	(*═════════════════════════════════════════════════════════*)
	(*  External Systems and I/O    *)
	(*═════════════════════════════════════════════════════════*)
	controlfb_control_b_start                                  , (* BOOL *)
	controlfb_control_b_stop                                   , (* BOOL *)
	controlfb_control_b_shutdown                               , (* BOOL *)
	controlfb_control_b_Reset                                  , (* BOOL *)
	controlfb_control_b_SystemShutdown                         , (* BOOL *)
	controlfb_control_b_EMstop                                 , (* BOOL *)
	controlfb_control_b_ClearHistory                           , (* BOOL *)
	controlfb_control_b_ActivateSettings                       , (* BOOL *)
	controlfb_control_b_startDeHum                             , (* BOOL *)
	controlfb_Operation_inputgrid_b_SyncClose                  , (* BOOL *)
	controlfb_Operation_Genset_b_manualStart                   , (* BOOL *)
	controlfb_Operation_PSB_b_SyncClose                        , (* BOOL *)
	controlfb_Operation_charger_b_StartCharging                , (* BOOL *)
	controlfb_Operation_charger_b_ResetCharger                 , (* BOOL *)
	controlfb_Operation_system_r_NominalVoltage                , (* REAL *)
	controlfb_Operation_system_r_NominalFrequency              , (* REAL *)
	controlfb_Operation_system_r_Pset                          , (* REAL *)
	controlfb_Operation_system_r_Qset                          , (* REAL *)
	controlfb_Operation_system_r_PFset                         , (* REAL *)
	controlfb_Operation_system_b_PFsetEnable                   , (* BOOL *)
	controlfb_Operation_system_b_SounderMute                   , (* BOOL *)
	controlfb_Operation_system_b_SounderTest                   , (* BOOL *)
	controlfb_Operation_system_b_GenGridModeTrans              , (* BOOL *)
	controlfb_Operation_system_b_GridTakeOverEnable            , (* BOOL *)
	controlfb_Operation_parallel_b_DetectSlaves                , (* BOOL *)
	controlfb_Operation_parallel_r_ActivePowerSlave1           , (* REAL *)
	controlfb_Operation_parallel_r_ReactivePowerSlave1         , (* REAL *)
	controlfb_Operation_parallel_r_ActivePowerSlave2           , (* REAL *)
	controlfb_Operation_parallel_r_ReactivePowerSlave2         , (* REAL *)
	controlfb_Operation_BMS_b_ManualStartHVDC                  , (* BOOL *)
	controlfb_SoftSettings_inputgrid_PeakshaveMode             , (* ePeakshaveMode *)
	controlfb_SoftSettings_inputgrid_setpointTimeslot1_r_SocTarget, (* REAL *)
	controlfb_SoftSettings_inputgrid_setpointTimeslot1_r_IdleChargePower, (* REAL *)
	controlfb_SoftSettings_inputgrid_setpointTimeslot1_r_FeedInCurrentLimitSoft, (* REAL *)
	controlfb_SoftSettings_inputgrid_setpointTimeslot1_r_SupplyCurrentLimitSoft, (* REAL *)
	controlfb_SoftSettings_inputgrid_setpointTimeslot2_r_SocTarget, (* REAL *)
	controlfb_SoftSettings_inputgrid_setpointTimeslot2_r_IdleChargePower, (* REAL *)
	controlfb_SoftSettings_inputgrid_setpointTimeslot2_r_FeedInCurrentLimitSoft, (* REAL *)
	controlfb_SoftSettings_inputgrid_setpointTimeslot2_r_SupplyCurrentLimitSoft, (* REAL *)
	controlfb_SoftSettings_inputgrid_b_BreakerControl          , (* BOOL *)
	controlfb_SoftSettings_inputgrid_b_ReverseCTDirection      , (* BOOL *)
	controlfb_SoftSettings_inputgrid_ui_CTrange                , (* UINT *)
	controlfb_SoftSettings_inputgrid_r_VTratio                 , (* REAL *)
	controlfb_SoftSettings_inputgrid_b_GridCodesActive         , (* BOOL *)
	controlfb_SoftSettings_inputgrid_b_WeakGridInput           , (* BOOL *)
	controlfb_SoftSettings_inputgrid_breaker_AutoConnect       , (* BOOL *)
	controlfb_SoftSettings_inputgrid_breaker_ShutdownDisconnect, (* BOOL *)
	controlfb_SoftSettings_inputgrid_breaker_EMstopDisconnect  , (* BOOL *)
	controlfb_SoftSettings_inputgrid_breaker_CurrentLimitDisconnect, (* BOOL *)
	controlfb_SoftSettings_inputgrid_breaker_CurrentLimitRetries, (* BYTE *)
	controlfb_SoftSettings_inputgenset_b_AutoStartStop         , (* BOOL *)
	controlfb_SoftSettings_inputgenset_b_HydridMode            , (* BOOL *)
	controlfb_SoftSettings_inputgenset_b_EnableSchedule        , (* BOOL *)
	controlfb_SoftSettings_inputgenset_setpointTimeslot1_r_SoCStart, (* REAL *)
	controlfb_SoftSettings_inputgenset_setpointTimeslot1_r_SoCStop, (* REAL *)
	controlfb_SoftSettings_inputgenset_setpointTimeslot1_r_BatteryloadStart, (* REAL *)
	controlfb_SoftSettings_inputgenset_setpointTimeslot1_r_BatteryloadStop, (* REAL *)
	controlfb_SoftSettings_inputgenset_setpointTimeslot1_b_StartAtBatteryError, (* BOOL *)
	controlfb_SoftSettings_inputgenset_setpointTimeslot2_r_SoCStart, (* REAL *)
	controlfb_SoftSettings_inputgenset_setpointTimeslot2_r_SoCStop, (* REAL *)
	controlfb_SoftSettings_inputgenset_setpointTimeslot2_r_BatteryloadStart, (* REAL *)
	controlfb_SoftSettings_inputgenset_setpointTimeslot2_r_BatteryloadStop, (* REAL *)
	controlfb_SoftSettings_inputgenset_setpointTimeslot2_b_StartAtBatteryError, (* BOOL *)
	controlfb_SoftSettings_inputgenset_b_PSBExtGensetMonitoring, (* BOOL *)
	controlfb_SoftSettings_inputgenset_b_FreqProtectionEnable  , (* BOOL *)
	controlfb_SoftSettings_inputgenset_Generator_e_GensetMode  , (* eGensetMode *)
	controlfb_SoftSettings_inputgenset_Generator_b_GensetLoadshareLine, (* BOOL *)
	controlfb_SoftSettings_inputgenset_Generator_r_RatedPower  , (* REAL *)
	controlfb_SoftSettings_inputgenset_Generator_r_powerloadMax, (* REAL *)
	controlfb_SoftSettings_inputgenset_Generator_r_PowerloadMin, (* REAL *)
	controlfb_SoftSettings_inputgenset_Generator_r_PowerloadEff, (* REAL *)
	controlfb_SoftSettings_inputgenset_Generator_r_ramprate    , (* REAL *)
	controlfb_SoftSettings_inputgenset_Generator_ui_CooldownTime, (* UINT *)
	controlfb_SoftSettings_inputgenset_Generator_ui_WarmupTime , (* UINT *)
	controlfb_SoftSettings_inputgenset_Loadbank_b_Enable       , (* BOOL *)
	controlfb_SoftSettings_inputgenset_Loadbank_r_PowerRating  , (* REAL *)
	controlfb_SoftSettings_inputgenset_Loadbank_r_PowerStepSize, (* REAL *)
	controlfb_SoftSettings_PSB_PeakshaveMode                   , (* ePeakshaveMode *)
	controlfb_SoftSettings_PSB_setpointTimeslot1_r_SocTarget   , (* REAL *)
	controlfb_SoftSettings_PSB_setpointTimeslot1_r_IdleChargePower, (* REAL *)
	controlfb_SoftSettings_PSB_setpointTimeslot1_r_FeedInCurrentLimitSoft, (* REAL *)
	controlfb_SoftSettings_PSB_setpointTimeslot1_r_SupplyCurrentLimitSoft, (* REAL *)
	controlfb_SoftSettings_PSB_setpointTimeslot2_r_SocTarget   , (* REAL *)
	controlfb_SoftSettings_PSB_setpointTimeslot2_r_IdleChargePower, (* REAL *)
	controlfb_SoftSettings_PSB_setpointTimeslot2_r_FeedInCurrentLimitSoft, (* REAL *)
	controlfb_SoftSettings_PSB_setpointTimeslot2_r_SupplyCurrentLimitSoft, (* REAL *)
	controlfb_SoftSettings_PSB_b_BreakerControl                , (* BOOL *)
	controlfb_SoftSettings_PSB_b_ReverseCTDirection            , (* BOOL *)
	controlfb_SoftSettings_PSB_ui_CTrange                      , (* UINT *)
	controlfb_SoftSettings_PSB_r_VTratio                       , (* REAL *)
	controlfb_SoftSettings_system_b_EnableSchedule             , (* BOOL *)
	controlfb_SoftSettings_system_b_EnableTransportMode        , (* BOOL *)
	controlfb_SoftSettings_system_b_EcoModeEnable              , (* BOOL *)
	controlfb_SoftSettings_system_e_UgridPowerMode             , (* eUgridPowerMode *)
	controlfb_SoftSettings_system_e_NetcontactorMode           , (* eNetcontMode *)
	controlfb_SoftSettings_system_e_UgridPowerLimitingMode     , (* ePLM *)
	controlfb_SoftSettings_system_b_AutomaticSwitching         , (* BOOL *)
	controlfb_SoftSettings_system_b_AMF                        , (* BOOL *)
	controlfb_SoftSettings_system_r_FrequencyDroop             , (* REAL *)
	controlfb_SoftSettings_system_r_VoltageDroop               , (* REAL *)
	controlfb_SoftSettings_system_r_SocMin                     , (* REAL *)
	controlfb_SoftSettings_system_r_SocMax                     , (* REAL *)
	controlfb_SoftSettings_system_r_PDischargeLimit            , (* REAL *)
	controlfb_SoftSettings_system_r_PChargeLimit               , (* REAL *)
	controlfb_SoftSettings_system_r_AMax                       , (* REAL *)
	controlfb_SoftSettings_system_s_SystemName                 , (* STRING(18) *)
	controlfb_SoftSettings_system_s_SMSnumber                  , (* STRING(18) *)
	controlfb_SoftSettings_system_ScheduleTimeSlot1_b_active   , (* BOOL *)
	controlfb_SoftSettings_system_ScheduleTimeSlot1_usi_DayOfWeek, (* USINT *)
	controlfb_SoftSettings_system_ScheduleTimeSlot1_usi_HourOfDay, (* USINT *)
	controlfb_SoftSettings_system_ScheduleTimeSlot1_usi_MinuteOfHour, (* USINT *)
	controlfb_SoftSettings_system_ScheduleTimeSlot2_b_active   , (* BOOL *)
	controlfb_SoftSettings_system_ScheduleTimeSlot2_usi_DayOfWeek, (* USINT *)
	controlfb_SoftSettings_system_ScheduleTimeSlot2_usi_HourOfDay, (* USINT *)
	controlfb_SoftSettings_system_ScheduleTimeSlot2_usi_MinuteOfHour, (* USINT *)
	controlfb_SoftSettings_system_by_LEDbrightness             , (* BYTE *)
	controlfb_SoftSettings_setup_e_AcInputType                 , (* eAcInputType *)
	controlfb_SoftSettings_setup_b_MasterSlaveMode             , (* BOOL *)
	controlfb_SoftSettings_setup_b_PeakshaveBoxEnable          , (* BOOL *)
	controlfb_SoftSettings_setup_e_Gridmode                    , (* eGridmode *)
	controlfb_SoftSettings_setup_e_DcCouplingType              , (* eDCinputType *)
	controlfb_SoftSettings_setup_b_ExtGenset                   , (* BOOL *)
	controlfb_HardSettings_setup_e_ControlSource               , (* eControlSources *)
	controlfb_HardSettings_charger_r_PowerMax                  , (* REAL *)
	controlfb_HardSettings_parallel_b_MasterSlaveEnabled       , (* BOOL *)
	controlfb_HardSettings_parallel_b_UnitIsMaster             , (* BOOL *)
	controlfb_HardSettings_parallel_b_ShutdownOnCommError      , (* BOOL *)
	controlfb_HardSettings_parallel_b_EffiencyMode             , (* BOOL *)
	controlfb_HardSettings_parallel_r_VoltageDroop             , (* REAL *)
	controlfb_HardSettings_parallel_r_FrequencyDroop           , (* REAL *)
	controlfb_HardSettings_system_r_PDischargeLimit            , (* REAL *)
	controlfb_HardSettings_system_r_PChargeLimit               , (* REAL *)
	controlfb_HardSettings_system_r_SMax                       , (* REAL *)
	controlfb_HardSettings_system_r_Amax                       , (* REAL *)
	controlfb_HardSettings_system_e_EarthingSystem             , (* eEarthingSystems *)
	controlfb_HardSettings_system_a_ui_InputCurrentLimit_1     , (* UINT *)
	controlfb_HardSettings_system_a_ui_InputCurrentLimit_2     , (* UINT *)
	controlfb_HardSettings_system_a_ui_OutputCurrentLimit_1    , (* UINT *)
	controlfb_HardSettings_system_a_ui_OutputCurrentLimit_2    , (* UINT *)
	controlfb_HardSettings_system_a_ui_OutputCurrentLimit_3    , (* UINT *)
	Generator_CommunicationOK                                  , (* BOOL *)
	Generator_FuelLow                                          , (* BOOL *)
	Generator_FuelCritical                                     , (* BOOL *)
	Generator_bGenBreakerClosed                                , (* BOOL *)
	Generator_bMainBreakerClosed                               , (* BOOL *)
	Generator_bGenRunning                                      , (* BOOL *)
	Generator_bGenVoltFreqOK                                   , (* BOOL *)
	Generator_bMainsFailure                                    , (* BOOL *)
	Generator_eActiveGenMode                                   , (* eGenOperationMode *)
	Generator_bIslandModeActive                                , (* BOOL *)
	Generator_bAMFActive                                       , (* BOOL *)
	Generator_bPeakshaveActive                                 , (* BOOL *)
	Generator_bFixedPowerActive                                , (* BOOL *)
	Generator_ar_LineVoltage_AVG                               , (* REAL *)
	Generator_ar_LineVoltage_L1                                , (* REAL *)
	Generator_ar_LineVoltage_L2                                , (* REAL *)
	Generator_ar_LineVoltage_L3                                , (* REAL *)
	Generator_ar_PhaseVoltage_AVG                              , (* REAL *)
	Generator_ar_PhaseVoltage_L1                               , (* REAL *)
	Generator_ar_PhaseVoltage_L2                               , (* REAL *)
	Generator_ar_PhaseVoltage_L3                               , (* REAL *)
	Generator_ar_Frequency_AVG                                 , (* REAL *)
	Generator_ar_Frequency_L1                                  , (* REAL *)
	Generator_ar_Frequency_L2                                  , (* REAL *)
	Generator_ar_Frequency_L3                                  , (* REAL *)
	Generator_ar_Current_AVG                                   , (* REAL *)
	Generator_ar_Current_L1                                    , (* REAL *)
	Generator_ar_Current_L2                                    , (* REAL *)
	Generator_ar_Current_L3                                    , (* REAL *)
	Generator_ar_PowerFactor_AVG                               , (* REAL *)
	Generator_ar_ActivePower_AVG                               , (* REAL *)
	Generator_ar_ActivePower_L1                                , (* REAL *)
	Generator_ar_ActivePower_L2                                , (* REAL *)
	Generator_ar_ActivePower_L3                                , (* REAL *)
	Generator_ar_ReactivePower_AVG                             , (* REAL *)
	Generator_ar_ApparentPower_AVG                             , (* REAL *)
	HartingIO_b_DigitalInput1Active                            , (* BOOL *)
	HartingIO_b_DigitalInput2Active                            , (* BOOL *)
	HartingIO_b_GenLowFuel                                     , (* BOOL *)
	HartingIO_b_ExtSystemShutdownRequest                       , (* BOOL *)
	HartingIO_b_ExtEMstopOK                                    , (* BOOL *)
	HartingIO_b_ExtEMstopActive                                , (* BOOL *)
	last
) DINT;
END_TYPE

// ---- POUs/MonitoringControl/IoT/DUTS/eIoTCommVersion.TcDUT
{attribute 'qualified_only'}
{attribute 'strict'}
TYPE eIoTCommVersion :
(
	V1 := 0,
	V2 := 1
);
END_TYPE

// ---- POUs/MonitoringControl/IoT/DUTS/eLogType.TcDUT
{attribute 'qualified_only'}
TYPE eLogType :
(
	none := 0,
	nuc := 1,
	cloud := 2
)UINT;
END_TYPE

// ---- POUs/MonitoringControl/IoT/DUTS/eUpdate.TcDUT
{attribute 'qualified_only'}
TYPE eUpdate :
(
	Fast			:= 0,
	Slow			:= 1,
	OnChange 		:= 2, //Updates only of variable has changed from previous value, but additionaly exactly once at system startup.
	Daily			:= 3
)UINT;
END_TYPE

// ---- POUs/MonitoringControl/IoT/DUTS/e_ORAttributeType.TcDUT
{attribute 'qualified_only'}
{attribute 'strict'}
TYPE e_ORAttributeType :
(
	text := 0,
	number := 2,
	integer := 3,
	JSON := 4
);
END_TYPE

// ---- POUs/MonitoringControl/IoT/DUTS/ST_AutoProvisioning.TcDUT
TYPE ST_AutoProvisioning :
	STRUCT
		sType	: STRING;
		sRealm	: STRING;
		sError	: STRING;
	END_STRUCT
END_TYPE

// ---- POUs/MonitoringControl/IoT/DUTS/ST_IotProps.TcDUT
TYPE ST_IotProps :
STRUCT
	sName		: STRING;
	sValue		: STRING(2000);
	eUpdate 	: eUpdate;
	st_RW		: ST_RW;
	pAdress		: PVOID;
	diSize		: DINT;
	ClassType : __SYSTEM.TYPE_CLASS;
	bNumber		: BOOL;
	bJson		: BOOL;
END_STRUCT
END_TYPE

// ---- POUs/MonitoringControl/IoT/DUTS/ST_RW.TcDUT
TYPE ST_RW :
STRUCT
	ReadFromNUC : BOOL:= FALSE;//enabling Read and Write can create unintended behaviour, consider feedback var
	WriteToNUC: BOOL:=FALSE ; //enabling Read and Write can create unintended behaviour, consider feedback var
END_STRUCT
END_TYPE

// ---- POUs/MonitoringControl/IoT/DUTS/ST_Supervisor.TcDUT
TYPE ST_Supervisor :
	STRUCT
		DATA	: STRING;
		ERROR	: STRING;
	END_STRUCT
END_TYPE

// ---- POUs/MonitoringControl/IoT/DUTS/ST_VarBuffer.TcDUT
TYPE ST_VarBuffer :
STRUCT
	sValue 	  : STRING(2000);
	pAdress   : PVOID;
	diSize	  : DINT;  
	ClassType : __SYSTEM.TYPE_CLASS;
	bNumber   : BOOL;
END_STRUCT
END_TYPE

// ---- POUs/MonitoringControl/IoT/_Structs/ST_IoTDataHMI.TcDUT
TYPE ST_IoTDataHMI :
STRUCT
	Label 				: STRING;
	Varname				: eDataMappingVarNames;
	Unit				: STRING(20);
	LogType 			: eLogType; 
	LogInterval 		: eUpdate;
	b_IOTWriteAllowed	: BOOL;
END_STRUCT
END_TYPE

// ---- POUs/MonitoringControl/IoT/_Structs/ST_IotData_credits.TcDUT
TYPE ST_IotData_credits :
STRUCT
	TotalCredits 		: DINT := 100;
	RemainingCredits	: DINT;
	UsedCredits			: DINT;
END_STRUCT
END_TYPE

// ---- POUs/MonitoringControl/IoT/_Structs/st_IOT_params.TcDUT
TYPE st_IOT_params :
STRUCT
	b_controlEnable			: 	BOOL := FALSE;
	r_UpdateTimeFast		: 	REAL := 15; //seconds
	r_UpdateTimeSlow		: 	REAL := 60; //seconds
	IotCommVersion			: 	eIotCommVersion;
	DefaultLoggingBudget	:	UINT	:= 100;
END_STRUCT
END_TYPE

// ---- POUs/MonitoringControl/IoT/_Structs/ST_IOT_SentStateLog.TcDUT
TYPE ST_IOT_SentStateLog :
STRUCT
	bUpdate			: BOOL;
	bMessageSent	: BOOL;
	LastIndexSent	: INT;
	LastIndex		: INT;
END_STRUCT
END_TYPE

// ---- POUs/MonitoringControl/_Enums/eAcInputType.TcDUT
{attribute 'qualified_only'}
{attribute 'strict'}
TYPE eAcInputType :
(
	None 	:= 0,
	Grid 	:= 1,
	Genset	:= 2
);
END_TYPE

// ---- POUs/MonitoringControl/_Enums/eCapTestSTate.TcDUT
{attribute 'qualified_only'}
{attribute 'strict'}
TYPE eCapTestSTate :
(
	init 				:= 	0,
	WriteSerial			:=	1,
	WriteNameplateCap	:=	2,
	WriteDatetime		:=	3,
	StartSystem 		:= 	4,
	InitialCharge 		:= 	5,
	RestPeriod1			:= 	6,
	DischargeCycle 		:= 	7,
	RestPeriod2 		:= 	8,
	ChargeCycle 		:= 	9,
	RestPeriod3 		:= 	10,
	StopSystem  		:= 	11,
	done				:=	12
);
END_TYPE

// ---- POUs/MonitoringControl/_Enums/eControlSources.TcDUT
{attribute 'qualified_only'}
{attribute 'strict'}
{attribute 'to_string'}
TYPE eControlSources :
(
	Local 				:= 0,
	ExternalController 	:= 1,
	PowerNet			:= 2	
);
END_TYPE

// ---- POUs/MonitoringControl/_Enums/eDcInputType.TcDUT
{attribute 'qualified_only'}
{attribute 'strict'}
TYPE eDcInputType :
(
	None := 0,
	Dc_charger := 1, 
	Dc_extender := 2
);
END_TYPE

// ---- POUs/MonitoringControl/_Enums/eEarthingSystems.TcDUT
{attribute 'qualified_only'}
{attribute 'strict'}
TYPE eEarthingSystems :
(
	None 		:= 0,	
	TN			:= 1,
	TN_ext		:= 2,
	IT			:= 3		
);
END_TYPE

// ---- POUs/MonitoringControl/_Enums/eGridFormingMode.TcDUT
{attribute 'qualified_only'}
{attribute 'strict'}
TYPE eGridFormingMode:
(
	Island := 0,
	Droop := 1
);
END_TYPE

// ---- POUs/MonitoringControl/_Enums/eGridMode.TcDUT
{attribute 'qualified_only'}
{attribute 'strict'}
{attribute 'to_string'}
TYPE eGridMode :
(
	auto := 0,
	following := 1,
	forming	:= 2
);
END_TYPE

// ---- POUs/MonitoringControl/_Enums/eNetContactorDirection.TcDUT
{attribute 'qualified_only'}
{attribute 'strict'}
TYPE eNetContactorDirection :
(
	Left 	:= -1,
	None 	:= 0,
	Right 	:= 1
);
END_TYPE

// ---- POUs/MonitoringControl/_Enums/eOperationMode.TcDUT
{attribute 'qualified_only'}
{attribute 'strict'}
TYPE eOperationMode :
(
	Auto := 0,
	Gridfollowing := 1,
	GridForming	:= 2
);
END_TYPE

// ---- POUs/MonitoringControl/_Enums/ePeakshaveMode.TcDUT
{attribute 'qualified_only'}
{attribute 'strict'}
TYPE ePeakshaveMode :
(
	Multiphase := 0,
	Singlephase := 1
);
END_TYPE

// ---- POUs/MonitoringControl/_Enums/ePowerControlType.TcDUT
{attribute 'qualified_only'}
{attribute 'strict'}
{attribue 'to_string}
TYPE ePowerControlType :
(
	Current := 0,
	Power	:=1,
	Both	:= 2
);
END_TYPE

// ---- POUs/MonitoringControl/_Enums/eSchedulerMode.TcDUT
{attribute 'qualified_only'}
{attribute 'strict'}
TYPE eSchedulerMode :
(
	continous := 0,
	daily := 1,
	weekly := 2
);
END_TYPE

// ---- POUs/MonitoringControl/_Enums/eSystemState.TcDUT
{attribute 'qualified_only'}
{attribute 'strict'}
{attribute 'to_string'}
TYPE eSystemState :
(
	Off 			:= 0,
	Shutdown 		:= 1,
	StandBy 		:= 2,
	Conditioning 	:= 3,
	Starting		:= 4,
	Running			:= 5,
	Charging_Only	:= 6,
	Discharging_Only:= 7,
	Stopped			:= 8,
	EMstop			:= 9,
	Reset			:= 10,
	Init			:= 11,
	Transport		:= 12,
	Dehumidifying	:= 13
);
END_TYPE

// ---- POUs/MonitoringControl/_Enums/eUgridPowerMode.TcDUT
{attribute 'qualified_only'}
{attribute 'strict'}
{attribute 'to_string'}
TYPE eUgridPowerMode :
(
	auto 			:= 0,
	DroopZeroStart	:= 1,
	Droop			:= 2,
	Isochronous		:= 3,
	None			:= 4
);
END_TYPE

// ---- POUs/MonitoringControl/_Structs/ST_ExtController_Events.TcDUT
TYPE ST_ExtController_Events :
STRUCT
	b_HeartbeatFault			: BIT;
	b_couplerError				:	bit;
	
	// control limit warnings
	b_FeedInLimitOutOfRange		: BIT;
	b_SupplyLimitOutOfRange 	: BIT;
	b_IdleChargePowerOutofRange	: BIT;
	b_BatOloadStartOutOfRange	: BIT;
	b_BatOloadStopOutOfRange	: BIT;
	b_SocTargetOutOfRange		: BIT;
	b_SocStartOutOfRange		: BIT;
	b_SocStopOutOfRange			: BIT;
	b_PsetOutOfRange			: BIT;
	b_QsetOutOfRange			: BIT;
	b_PFsetOutOfRange			: BIT;
	b_NominalVoltageOutOfRange	: BIT;
	b_NominalFreqOutOfRange		: BIT;
	b_FreqDroopOutOfRange		: BIT;
	b_VoltageDroopOutOfRange	: BIT;
	b_PmaxOutOfRange			: BIT;
	b_PminOutOfRange			: BIT;
	b_SmaxOutOfRange			: BIT;
	b_AmaxOutOfRange			: BIT;
	b_PowerRamprateOutOfRange	: BIT;
	b_PSBFeedInLimitOutOfRange	: BIT;
	b_PSBSupplyLimitOutOfRange: BIT;
	b_PSBIdleChargePowerOutOfRange: BIT;
	b_PSBSoCTargetOutOfRange	: BIT;
	b_SoCHighLimitOutOfRange	: BIT;
	b_SoCLowLimitOutOfRange		: BIT;
	b_GridModeValueOutOfRange	: BIT;
	b_PowermodeValueOutOfRange	: BIT;

END_STRUCT
END_TYPE

// ---- POUs/MonitoringControl/_Structs/ST_ExtController_get.TcDUT
TYPE ST_ExtController_get :
STRUCT
	control							: ST_ControlVars;
	Operation						: ST_OperationVars;
	SoftSettings					: ST_SoftSettings;
	HardSettings					: ST_HardSettings;
	events							: ST_ExtController_Events;
	b_AdvancedControl				: BOOL;
	ui_Heartbeat					: UINT;
	s_dashboardID					: STRING;
	b_Active						: BOOL;
	e_ConnectionState				: eConnectionState;
	s_OutputJson					: STRING(2000);
	LoggingBudgetOK					: BOOL := TRUE;
END_STRUCT
END_TYPE

// ---- POUs/MonitoringControl/_Structs/ST_ExtController_limits.TcDUT
TYPE ST_ExtController_limits :
STRUCT
	r_InputCtLimit			: REAL := 800;
	r_InverterPowerLimit	: REAL := 360;
	r_InverterCurrentLimit	: REAL := 520;
	r_NominalVoltageMin		: REAL := 360;
	r_NominalVoltageMax		: REAL := 440;
	r_NominalFreqMin		: REAL := 47.5;
	r_NominalFreqMax		: REAL := 52.5;
	r_DroopMax				: REAL := 10; 
	r_PowerRampLimit		: REAL := 300; //%/s
	r_PSBCtLimit			: REAL := 4000;
END_STRUCT
END_TYPE

// ---- POUs/MonitoringControl/_Structs/ST_ExtController_Set.TcDUT
TYPE ST_ExtController_Set :
STRUCT
	b_available				: BOOL;
END_STRUCT
END_TYPE

// ---- POUs/MonitoringControl/_Structs/ST_PLCPersistentVars.TcDUT
TYPE ST_PLCPersistentVars :
STRUCT
	Hardsettings					: ST_HardSettings; 
	Softsettings					: ST_Softsettings;
END_STRUCT
END_TYPE

// ---- POUs/Objects/4Grouter/Struct/ST_router_service.TcDUT
TYPE ST_router_service :
STRUCT
END_STRUCT
END_TYPE

// ---- POUs/Objects/ACDCCharger/Structs/ST_ACDCCharger_Service.TcDUT
TYPE ST_ACDCCharger_Service :
STRUCT
END_STRUCT
END_TYPE

// ---- POUs/Objects/BMS/eNums/eBMS_Status.TcDUT
{attribute 'qualified_only'}
{attribute 'strict'}
{attribute 'to_string'} 
TYPE eBMS_Status :
(
	Init := 0,
	Normal := 1,
	FullCharge := 2,
	FullDischarge := 3,
	Warning := 4,
	Fault := 5,
	off := 6
);
END_TYPE

// ---- POUs/Objects/BMS/eNums/eHVDC_Powerstatus.TcDUT
{attribute 'qualified_only'}
{attribute 'strict'}
TYPE eHVDC_Powerstatus :
(
	OFF := 0,
	Precharging := 1,
	ON	:= 2	
);
END_TYPE

// ---- POUs/Objects/BMS/eNums/ePOUState.TcDUT
{attribute 'qualified_only'}
{attribute 'strict'}
TYPE ePOUState :
(
	OFF := 0,
	PowerUp := 1,
	Init := 2,
	Normal	:=	3,
	EMSTOP	:=	4,
	Shutdown := 5
);
END_TYPE

// ---- POUs/Objects/BMS/eNums/ePowerControl.TcDUT
{attribute 'qualified_only'}
{attribute 'strict'}
TYPE ePowerControl :
(
	Init := 0,
	Stay := 1,
	PowerOn := 2,
	PowerOff := 3
)word;
END_TYPE

// ---- POUs/Objects/BMS/eNums/ePowerOnStatus.TcDUT
{attribute 'qualified_only'}
{attribute 'strict'}
TYPE ePowerOnStatus :
(
	Off := 0,
	On	:= 1,
	PowerOn_Fault := 2,
	PowerOff_Fault := 3
)UINT;
END_TYPE

// ---- POUs/Objects/BMS/Structs/st_BMS_BatterySummary.TcDUT
TYPE st_BMS_BatterySummary EXTENDS st_MBMU_BatterySummary :
STRUCT
	r_ratedPower				: REAL;
	r_ratedCurrent				: REAL;
	r_ratedEnergyCapacity		: REAL;
	ui_CycleCount				: UINT;
	r_SOCScaled					: REAL;
	b_chargingAllowed			: BOOL;
	b_dischargingAllowed		: BOOL;
	r_RemainingDischargeEnergyNett: REAL;
	r_RemainingChargeEnergyNett	: REAL;
	r_maxVoltageEver	 		: REAL;
	r_maxChargeCurrentEver		: REAL;
	r_maxDischargeCurrentEver	: REAL;
END_STRUCT
END_TYPE

// ---- POUs/Objects/BMS/Structs/st_BMS_Events.TcDUT
TYPE st_BMS_Events :
STRUCT
	//sunspec error list
	b_COMMUNICATION_ERROR			:	BOOL;
	b_OVER_TEMP_ALARM				:	BOOL;
	b_OVER_TEMP_WARNING				:	BOOL;
	b_UNDER_TEMP_ALARM				:	BOOL;
	b_UNDER_TEMP_WARNING			:	BOOL;
	b_OVER_CHARGE_CURRENT_ALARM		:	BOOL;
	b_OVER_CHARGE_CURRENT_WARNING	:	BOOL;
	b_OVER_DISCHARGE_CURRENT_ALARM	:	BOOL;
	b_OVER_DISCHARGE_CURRENT_WARNING:	BOOL;
	b_OVER_VOLT_ALARM				:	BOOL;
	b_OVER_VOLT_WARNING				:	BOOL;
	b_UNDER_VOLT_ALARM				:	BOOL;
	b_UNDER_VOLT_WARNING			:	BOOL;
	b_UNDER_SOC_MIN_ALARM			:	BOOL;
	b_UNDER_SOC_MIN_WARNING			:	BOOL;
	b_OVER_SOC_MAX_ALARM			:	BOOL;
	b_OVER_SOC_MAX_WARNING			:	BOOL;
	b_VOLTAGE_IMBALANCE_WARNING		:	BOOL;
	b_TEMPERATURE_IMBALANCE_ALARM	:	BOOL;
	b_TEMPERATURE_IMBALANCE_WARNING	:	BOOL;
	b_CONTACTOR_ERROR				:	BOOL;
	b_FAN_ERROR						:	BOOL;
	b_GROUND_FAULT					:	BOOL;
	b_OPEN_DOOR_ERROR				:	BOOL;
	b_CURRENT_IMBALANCE_WARNING		:	BOOL;
	b_OTHER_ALARM					:	BOOL;
	b_OTHER_WARNING					:	BOOL;
	b_CONFIGURATION_ALARM			:	BOOL;
	b_CONFIGURATION_WARNING			:	BOOL;
	b_POWERONFAULT					: 	BOOL;
	b_POWEROFFFAULT					:	BOOL;
	b_DISCONNECTOR_OFF				: 	BOOL;
	
	b_SocLowLimitOutOfRange			:	BOOL;
	b_SocHighLimitOutOfRange		: 	BOOL;
	
	b_SBMUCommError					:	ARRAY [0..3] OF BOOL;	
	b_SBMUFailedToConnect			:	ARRAY [0..3] OF BOOL;

	(* old event list. Replaced by sunspec
	BMSWatchdogWarning				:	BOOL;
	BMSWatchdogError				:	BOOL;
	
	BMSWarningStatus				:	BOOL;
	BMSFaultStatus					:	BOOL;
	
	BMSPowerOnFault					:	BOOL;
	BMSPowerOffFault				:	BOOL;
	
	SOCLowWarning					: 	BOOL;
	OverVoltageWarning				:	BOOL;
	UnderVoltageWarning				:	BOOL;
	VoltageBalanceWarning			:	BOOL;
	
	OverTemperatureWarning			:	BOOL;
	UnderTemperatureWarning			:	BOOL;
	TemperatureDifferenceWarning	:	BOOL;
	
	OverCurrentWarning				:	BOOL;
	
	CommunicationWarning			:	BOOL;
	
	OverVoltageError				:	BOOL;
	UnderVoltageError				:	BOOL;
	OverTemperatureError			:	BOOL;
	UnderTemperatureError			:	BOOL;
	
	CSCError						:	BOOL;
	SBMUError						:	BOOL;
	MBMUError						:	BOOL;
	
	CommunicationError				:	BOOL;
	*)
END_STRUCT
END_TYPE

// ---- POUs/Objects/BMS/Structs/st_BMS_Get.TcDUT
TYPE st_BMS_Get :
STRUCT
	BatteryInfo					: st_BMS_BatterySummary;
	t_RemainingTimeToAutoCalibration : TIME;
	//detailed info	
	MBMU						:	st_MBMU_Status;
	SBMU						:	ARRAY[0..3] OF st_SBMU_Status;
	
	Events						:	st_BMS_Events;
END_STRUCT
END_TYPE

// ---- POUs/Objects/BMS/Structs/st_BMS_Params.TcDUT
TYPE st_BMS_Params :
STRUCT
	IP_BMS							:	STRING(16) := '192.168.1.60';
	r_SocHysteresis					:   REAL := 1; // % 
	r_InternalConditioningSoCMin	: 	REAL := 30;
	r_SoCAbsoluteMin				: 	REAL := 6; // unscaled value
	r_SoCAbsoluteMax				: 	REAL := 100; //unscaled value

	r_KwhperString					: REAL := 208; //
	r_CrateBattery					: REAL := 0.5; //C
	r_AhperString					: REAL := 306; //Ah	
	b_DisableSOCAlarm				: BOOL := FALSE;
	b_ResetPersistentVars			: BOOL := FALSE;
	b_forcePrecharging				: BOOL := FALSE;
	
	b_EnableAutoCalibration			: BOOL := TRUE;
	t_AutoCalibrationInterval 		: TIME := T#14D;
END_STRUCT
END_TYPE

// ---- POUs/Objects/BMS/Structs/ST_BMS_Service.TcDUT
TYPE ST_BMS_Service :
STRUCT
END_STRUCT
END_TYPE

// ---- POUs/Objects/BMS/Structs/st_BMS_Set.TcDUT
TYPE st_BMS_Set :
STRUCT
	b_enable	: BOOL := TRUE;
	r_SocMax	: REAL := 90;
	r_SocMin	: REAL := 10;
END_STRUCT
END_TYPE

// ---- POUs/Objects/BMS/Structs/st_MBMU_BatterySummary.TcDUT
TYPE st_MBMU_BatterySummary :
STRUCT
		//general
	b_BMSHeartBeatOK				:	BOOL;
	e_BMS_PowerOnStatus				:	ePowerOnStatus;
	e_BMS_Status					:	eBMS_Status;		

	r_SystemVoltage					:	REAL;
	r_SystemCurrent					:	REAL;
	r_SOC							:	REAL;
	r_SOH							:	REAL := 100;
	ar_CellVoltage					:	ARRAY[0..2] OF REAL;
	ar_CellTemperature				:	ARRAY[0..2] OF REAL;
	r_MaxChargeCurrentAllowed		:	REAL;
	r_MaxDischargeCurrentAllowed	:	REAL;
	r_MaxChargePowerAllowed			:	REAL;
	r_MaxDischargePowerAllowed		:	REAL;
	r_MaxSystemVoltageAllowed		:	REAL;
	r_MinSystemVoltageAllowed		:	REAL;
	
	r_SystemPower					:	REAL;
	r_ChargeSOE						:	REAL;
	r_DischargeSOE					:	REAL;
	
	r_RemainingChargeEnergy			:	REAL;
	r_RemainingDischargeEnergy		:	REAL;
	
	r_HistAccChargeEnergy			:	REAL;
	r_HistAccDischargeEnergy		:	REAL;
END_STRUCT	
END_TYPE

// ---- POUs/Objects/BMS/Structs/st_MBMU_Status.TcDUT
TYPE st_MBMU_Status :
STRUCT
	GeneralSBMUStatus			:	ARRAY [0..15] OF WORD;
	MBMUStatus					:	ARRAY [0..15] OF WORD;

	s_MBMU_SWVer				:	STRING(16);
	s_MBMU_HWVer				:	STRING(16);
	
	s_ETH_SWVer					:	STRING(32);
	r_ETH_HWVer					:	STRING(32);	
	
	by_NumberOfSubSystems		:	BYTE;
	DateTime					:	ARRAY[0..5] OF WORD;
	b_InsulationSwitchOpen		:	BOOL;
	
	BatteryStatus				:	st_MBMU_BatterySummary;
END_STRUCT
END_TYPE

// ---- POUs/Objects/BMS/Structs/st_SBMU_BatterySummary.TcDUT
TYPE st_SBMU_BatterySummary :
STRUCT
	r_SystemVoltage			:	REAL;
	r_SystemCurrent			:	REAL;
	r_SOC					:	REAL;
	r_SOH					:	REAL;
	ar_CellVoltage				:	ARRAY[0..2] OF REAL;
	ar_CellTemperature			:	ARRAY[0..2] OF REAL;
	r_MaxChargeCurrentAllowed		:	REAL;
	r_MaxDischargeCurrentAllowed	:	REAL;
	r_HistAccChargeEnergy			:	REAL;
	r_HistAccDischargeEnergy		:	REAL;
	
	//Gaan we hier uberhaupt iets mee doen?
	w_MaxVoltageCellLocation 	: 	WORD;//ARRAY[0..1] OF BYTE;
	w_MinVoltageCellLocation 	:	 WORD;//ARRAY[0..1] OF BYTE;
	w_MaxTempCellLocation 		: 	WORD;//ARRAY[0..1] OF BYTE;
	w_MinTempCellLocation 		: 	WORD;//ARRAY[0..1] OF BYTE;
END_STRUCT
END_TYPE

// ---- POUs/Objects/BMS/Structs/st_SBMU_Status.TcDUT
TYPE st_SBMU_Status :
STRUCT
	w_SystemWarning			:	WORD;
	SystemAlarm				:	ARRAY [0..2] OF WORD;
	
	b_PrechargeRelayClosed	:	BOOL;
	b_MainPosRelayClosed	:	BOOL;
	b_MainNegRelayClosed	:	BOOL;
	b_ControlBoxFanOn		:	BOOL;
	b_BalanceStatus			:	BOOL;
	b_DoorState				:	BOOL;	
	
	s_SBMU_SWVer			:	STRING(16);
	s_SBMU_HWVer			:	STRING(16);
	s_CSC_SWVer				:	STRING(16);
	s_CSC_HWVer				:	STRING(16);
	
	BatteryStatus			:	st_SBMU_BatterySummary;
END_STRUCT
END_TYPE

// ---- POUs/Objects/CoolingSystem/enums/eConditioningRequirement.TcDUT
{attribute 'qualified_only'}
{attribute 'strict'}
{attribute 'to_string'}
TYPE eConditioningRequirement :
(
	none := 0,
	Pumprequired		:=	1,
	HeatingRequired 	:= 	2,
	CoolingRequired 	:= 	3
);
END_TYPE

// ---- POUs/Objects/CoolingSystem/enums/eCoolingSystemState.TcDUT
{attribute 'qualified_only'}
{attribute 'strict'}
{attribute 'to_string'}
TYPE eCoolingSystemState :
(
	OFF 						:= 	0,
	Circulating					:=	1,
	ActiveCooling				:= 	2,
	ActiveHeating				:= 	3,
	EMSTOP						:=	5
)uint := OFF;
END_TYPE

// ---- POUs/Objects/CoolingSystem/enums/eHeatPumpMode.TcDUT
{attribute 'qualified_only'}
{attribute 'strict'}
{attribute 'to_string'}
TYPE eHeatPumpMode :
(
	Standby := 0,
	Cooling := 1,
	Heating := 2
)UINT := Standby;
END_TYPE

// ---- POUs/Objects/CoolingSystem/enums/eHeatPumpState.TcDUT
{attribute 'qualified_only'}
{attribute 'strict'}
{attribute 'to_string'}
TYPE eHeatPumpState :
(
	OFF := 0,
	Initializing := 1,
	Standby := 2,
	Active_Cooling := 3,
	Active_Heating := 4,
	ERROR := 5
)UINT := OFF;
END_TYPE

// ---- POUs/Objects/CoolingSystem/enums/eSupportedHeatpumps.TcDUT
{attribute 'qualified_only'}
{attribute 'strict'}
TYPE eSupportedHeatpumps :
(
	TranePicco := 0,
	LgThermaV	:= 1
);
END_TYPE

// ---- POUs/Objects/CoolingSystem/structs/LG_Coils.TcDUT
TYPE LG_Coils :
STRUCT
	b_EnableOperation			:	BOOL := FALSE;
	b_EnableSwwOperation		: 	BOOL := FALSE;
	b_EnableSilentMode			:	BOOL := FALSE;
	b_EnableDesinfectionMode	:	BOOL := FALSE;
	b_EmstopActive				:	BOOL := FALSE;
	b_EnableEmStop				:	BOOL := FALSE;
END_STRUCT
END_TYPE

// ---- POUs/Objects/CoolingSystem/structs/LG_ControlRegs.TcDUT
TYPE LG_ControlRegs :
STRUCT
	ui_OperatingMode	:	UINT := 3;
	ui_ControlMode		:	UINT := 1;
	r_Setpoint1			:	REAL := 20;
	r_RoomSetpoint		:	REAL;
	ui_TempShiftValue	:	UINT;
	r_setpoint2			:	REAL;
	r_RoomSetpoint2		:	REAL;
	ui_TempShiftValue2	:	UINT;
	r_DHWgoalTemp		:	REAL;
	ui_EnergyStatus		:	UINT := 2;	
END_STRUCT
END_TYPE

// ---- POUs/Objects/CoolingSystem/structs/LG_InputRegs.TcDUT
TYPE LG_InputRegs :
STRUCT
	UI_ErrorCode		:	UINT;
	ui_OperationalMode	:	UINT;
	r_CoolantInletTemp	:	REAL;
	r_CoolantOutletTemp	:	REAL;
	r_BackupHeaterTemp	:	REAL;
	r_SWWTankTemp		:	REAL;
	r_SolarCollectorTemp:	REAL;
	r_RoomTemp1			:	REAL;
	r_FlowRate			:	REAL;
	r_FlowTempCircuit2	:	REAL;
	r_RoomTemp2			:	REAL;
	UI_EnergyStatus		:	UINT;
	r_OutsideTemp		:	REAL;	
	r_CoolantPressure	: Real;
END_STRUCT
END_TYPE

// ---- POUs/Objects/CoolingSystem/structs/LG_Statusbits.TcDUT
TYPE LG_Statusbits :
STRUCT
	b_WaterFlowNOK				:	BOOL;
	b_WaterPumpOn				:	BOOL;
	b_ExtWaterPumpOn			:	BOOL;
	b_CompressorOn				:	BOOL;
	b_DefrostOn					:	BOOL;
	b_SWWModeOn					:	BOOL;
	b_SWWTankDesinfectionActive	:	BOOL;
	b_SilentModeOn				:	BOOL;
	b_CoolingActive				:	BOOL;
	b_SolarPumpActive			:	BOOL;
	b_BackupHeater1Active		:	BOOL;
	b_BackupHeater2Active		:	BOOL;
	b_SWWBoostHeaterActive		:	BOOL;
	b_ErrorActive				:	BOOL;
	b_EMOperationAvailable		:	BOOL;
	b_EMSWWOperationAvailable	:	BOOL;
	b_MixPumpActive				:	BOOL;
	
END_STRUCT
END_TYPE

// ---- POUs/Objects/CoolingSystem/structs/ST_CoolingSystem_Events.TcDUT
TYPE ST_CoolingSystem_Events :
STRUCT
	//faults
	b_CoolingSystemFuseFailure		: 	BOOL;
	
	
	//System pressure dropped below idle minimum pressure. suspect coolant loss.
	b_CoolingLoopPressureLow	: 	BOOL := FALSE;	
	b_CoolingLoopPressureTooLow	: 	BOOL := FALSE;	
	
	//Temperature errors
	b_CoolantTempLow				: 	BOOL;
	b_CoolantTempTooHigh			: 	BOOL;
	b_CoolantTempHigh				: 	BOOL;
	
	HeatpumpEvents					:	ST_HeatpumpEvents;
END_STRUCT
END_TYPE

// ---- POUs/Objects/CoolingSystem/structs/ST_CoolingSystem_Get.TcDUT
TYPE ST_CoolingSystem_Get :
STRUCT
	CoolingSystemState		:	eCoolingSystemState;
	HeatPumpStatus			: 	eHeatPumpState;
	r_CoolantTemperature	:	REAL;
	r_CoolantPressure		:	REAL;
	r_EnclosureDewpoint		:	REAL;
	ui_DehumRemainingTime	: 	UINT; //minutes
	
	Heatpump			:	st_Heatpump_get;
	
	Events					: ST_CoolingSystem_Events;
END_STRUCT
END_TYPE

// ---- POUs/Objects/CoolingSystem/structs/ST_CoolingSystem_MaintenanceParams.TcDUT
TYPE ST_CoolingSystem_MaintenanceParams :
STRUCT
	//manual activation of cooling system. Max runtime is limited to 30 minutes
	b_ActivateCooling							: BOOL; 
	b_ActivateHeating							: BOOL;	
	
	
END_STRUCT
END_TYPE

// ---- POUs/Objects/CoolingSystem/structs/ST_Coolingsystem_params.TcDUT
TYPE ST_Coolingsystem_params :
STRUCT
	b_DoubleHeatpump							: BOOL := FALSE;
	
	// Minimum base coolant pressure
	r_MinimumSystemBasePressureWarningLevel		: REAL := 1;
	r_MinimumSystemBasePressureErrorLevel		: REAL := 0.7;

	PrimaryHeatpumpAddr							:	BYTE := 1;
	CoilSettings								:	BYTE := 2#0000_0001;
	SecondaryHeatpumpAddr						:	BYTE := 2;
	dw_HeatpumpOperationDelay					: DWORD := 30; // minutes
	
	//If the heatpump has run within this timeframe, no preheating is required before operation can start
	i_SkipHPPreheatingTime						: 	INT		:= 60; //minutes. 
	r_MinimumCoolantTemperatureForHPHeatingMode	:	REAL	:= 15;
	
	IO_IPaddress								: 	STRING := '192.168.1.52';
END_STRUCT
END_TYPE

// ---- POUs/Objects/CoolingSystem/structs/ST_HeatpumpData.TcDUT
TYPE ST_HeatpumpData :
STRUCT
	i_FW_Version		:	INT;		//1
	i_FW_release		:	INT;		//2
	w_FW_Subrelease		:	WORD;		//3
	w_FW_creationDate	:	WORD;		//4
	
	w_Serialnumber		:	ARRAY[0..17] OF WORD;	//80-97
	
	i_OperatingHours	:	INT;		//305-317?
	
	r_CoolantPower		:  	REAL;
	r_InletWaterTemp	:	REAL;		//400
	r_OutletWaterTemp	:	REAL;		//401
	r_HighPressure		:	REAL;		//406
	r_LowPressure		:	REAL;		//414
	r_CompInputTemp		:	REAL;		//422
	r_OutdoorTemp		:	REAL;		//428
	r_CompOutputTemp	:	REAL;		//433-435
	ui_WaterFlowRate		:	UINT;		//444
	
	w_ErrorList			:	ARRAY[1..7] OF WORD;	//950-956	
	
	r_FanSpeedPCT		:	REAL;		//7000
	r_PumpSpeedPCT		:	REAL;		//7001
	
	r_SetpointHeating	:	REAL;		//7204
	r_SetpointCooling	:	REAL;		//7203
	b_DefrostingActive	:	BOOL;		//7214.14
	
	HeatpumpEvents		:	st_HeatpumpEvents;
END_STRUCT
END_TYPE

// ---- POUs/Objects/CoolingSystem/structs/ST_HeatPumpEvents.TcDUT
TYPE ST_HeatPumpEvents :
STRUCT
	b_CommWarning		: BOOL;
	b_ProbeError		: BOOL;
	b_PressureError		: BOOL;
	b_CompressorError	: BOOL;
	b_ValveError		: BOOL;
	b_FanError			: BOOL;
	b_PumpError			: BOOL;
	b_WaterTempError	: BOOL;
	b_IOError			: BOOL;
	b_DefrostingActive	:	Bool;
	b_HeatpumpPreheatingActive	:	BOOL;
	b_TooColdForHeatpumpHeating	:	Bool;
END_STRUCT
END_TYPE

// ---- POUs/Objects/CoolingSystem/structs/ST_HeatPump_Get.TcDUT
TYPE ST_HeatPump_Get :
STRUCT
	HeatPumpState 	: 	eHeatPumpState;
	Setpoint		:	REAL;
	Events			: 	ST_HeatPumpEvents;
	
	HeatpumpData	:	ST_HeatpumpData;
END_STRUCT
END_TYPE

// ---- POUs/Objects/CoolingSystem/structs/st_TCME31_get_1.TcDUT
TYPE st_TCME31_get_1 :
STRUCT
	DigitalInput1	:	Bool;
	DigitalInput2	:	Bool;
	
	AnalogInput1	:	real;
	AnalogInput2	:	real;

	DigitalOutput1	:	Bool;
	DigitalOutput2	:	Bool;
	DigitalOutput3	:	Bool;
	DigitalOutput4	:	Bool;
	
	b_CommFault		:	Bool;
END_STRUCT
END_TYPE

// ---- POUs/Objects/CoolingSystem/structs/st_TCME31_Set_1.TcDUT
TYPE st_TCME31_Set_1 :
STRUCT
	IPAddress		:	String := '192.168.1.70';
	
	DigitalOutput1	:	Bool;
	DigitalOutput2	:	Bool;
	DigitalOutput3	:	Bool;
	DigitalOutput4	:	Bool;
END_STRUCT
END_TYPE

// ---- POUs/Objects/DCLink/_Enums/eDcLinkState.TcDUT
{attribute 'qualified_only'}
{attribute 'strict'}
{attribute 'to_string'} 

TYPE eDcLinkState :
(
	Disabled 	:= 0,
	Enabled	 	:= 1,
	Fault	 	:= 2
);
END_TYPE

// ---- POUs/Objects/DCLink/_Enums/eDCpowerPriority.TcDUT
{attribute 'qualified_only'}
{attribute 'strict'}
TYPE eDCpowerPriority :
(
	auto := 0,
	Inverter := 1,
	DCcoupling	:= 2
);
END_TYPE

// ---- POUs/Objects/DCLink/_Structs/ST_Bourns_errors.TcDUT
TYPE ST_Bourns_errors :
STRUCT
	b_OvervoltageError		:	BOOL;
	b_OverCurrentError		:	BOOL;
	b_OverTemperatureError	:	BOOL; 
	b_EnergyOverflow		:	BOOL;
	b_DeviceFault			:	BOOL;
	b_CommFault				:	BOOL;
END_STRUCT
END_TYPE

// ---- POUs/Objects/DCLink/_Structs/ST_Bourns_Powerdata.TcDUT
TYPE ST_Bourns_Powerdata :
STRUCT
	Power			: REAL;
	Current			: REAL;
	Voltage			: REAL;
	Energy			: REAL;
	EnergyImport	: REAL;
	EnergyExport	: REAL;
	Temperature		: REAL;
	Charge			: BOOL;
END_STRUCT
END_TYPE

// ---- POUs/Objects/DCLink/_Structs/ST_DCLink_events.TcDUT
TYPE ST_DCLink_events :
STRUCT
	OvercurrentTrip			: BOOL;
	OvervoltageNOK			: BOOL;
END_STRUCT
END_TYPE

// ---- POUs/Objects/DCLink/_Structs/ST_DCLink_Get.TcDUT
TYPE ST_DCLink_Get :
STRUCT
	b_DCCouplingState				: BOOL;
	Powerdata						: REFERENCE TO ST_Bourns_Powerdata;
	r_ratedCurrent					: REAL;
	r_BattChargePowerLimit			: REAL;
	r_BattDischargePowerLimit		: REAL;
	
	r_ExportPowerLimit				: REAL;
	r_ExportCurrentLimit			: REAL;
	r_ImportPowerLimit				: REAL;
	r_ImportCurrentLimit			: REAL;
	events							: ST_DCLink_events;
END_STRUCT
END_TYPE

// ---- POUs/Objects/DCLink/_Structs/ST_DCLink_IO.TcDUT
TYPE ST_DCLink_IO :
STRUCT
	bMCCBOpen		AT %Q*: BOOL;
	bMCCBClose		AT %Q*: BOOL;
	bUVRfb			AT %I*: BOOL;
END_STRUCT
END_TYPE

// ---- POUs/Objects/DCLink/_Structs/ST_DCLink_params.TcDUT
TYPE ST_DCLink_params :
STRUCT
	RatedCurrent			: UINT 		:= 250;
	OvercurrentTripDelay	: TIME		:= T#2S;
	IP						: STRING 	:= '192.168.1.62';
	DCpowerControlHyst		: REAL 		:= 0.1;	
	AllowClosingOnDeadBus	:	BOOL	:= FALSE;
	DIWiredToPLC			:	BOOL	:=	TRUE;
END_STRUCT
END_TYPE

// ---- POUs/Objects/DCLink/_Structs/ST_DCLink_set.TcDUT
TYPE ST_DCLink_set :
STRUCT
	b_DCBusEnable			:	Bool;
//	b_MCCBclose				: BOOL;
//	b_MCCBopen				: BOOL;
	r_ChargePowerLimit		: REAL;
	r_DischargePowerLimit	: REAL;
	r_DCCRatedPower			: REAL; // of the external device
	r_PowerRampRate			: REAL;
	e_DCpowerPriority		: eDCpowerPriority := eDCpowerPriority.DCcoupling;
END_STRUCT
END_TYPE

// ---- POUs/Objects/DCLink/_Structs/st_Pixsys.TcDUT
TYPE st_Pixsys :
STRUCT
	b_DoEnable			: BOOL;	
	b_DoFeedbackOn 		: BOOL;
	b_Di1				: BOOL;
	b_Di2				: BOOL;		
END_STRUCT
END_TYPE

// ---- POUs/Objects/PowerQualityMonitor/_Enums/eACRotationState.TcDUT
{attribute 'qualified_only'}
{attribute 'strict'}
{attribute 'to_string'}
TYPE eACRotationState :
(
	Left := -1,
	None := 0,
	Right := 1
);
END_TYPE

// ---- POUs/Objects/PowerQualityMonitor/_Structs/ST_PowerMonitor_BESS.TcDUT
TYPE ST_PowerMonitor_BESS :
STRUCT
	e_ACrotationStatus			: 	eACrotationState;
	ar_Current					:	ARRAY [0..4] OF REAL;
	r_LineVoltage				: 	REAL;
	r_Frequency					: 	REAL;
	r_currentUnbalance			:	REAL;
	//Power
	r_ApparentPower				: 	REAL;
	r_ReactivePower				: 	REAL;
	r_ActivePower				: 	REAL;
	//Energy Consumed
	r_EnergyConsumed			:	REAL;
	
	//Energy Delivered
	r_EnergySupplied			:	REAL;
	
	r_PowerFactor 				:	REAL;
END_STRUCT
END_TYPE

// ---- POUs/Objects/PowerQualityMonitor/_Structs/ST_PowerMonitor_Events.TcDUT
TYPE ST_PowerMonitor_Events :
STRUCT
	b_MBCommWarning 		: BOOL;
	b_MBCommError 			: BOOL;
	b_MBTimeoutWarning 		: BOOL;
	b_EL3443Warning			: BOOL;
	b_EL3443Error		: BOOL;
	b_ACdirectionDataInvalid: BOOL;
END_STRUCT
END_TYPE

// ---- POUs/Objects/PowerQualityMonitor/_Structs/ST_PowerMonitor_get.TcDUT
TYPE ST_PowerMonitor_get :
STRUCT
	InputField			:	ST_PowerMonitor_InputField;	
	OutputField			:	ST_PowerMonitor_OutputField;
	CEE					:   ST_PQVoltageData;
	Inverter			: 	ST_PQVoltageData;
	events				:	ST_PowerMonitor_Events;
END_STRUCT
END_TYPE

// ---- POUs/Objects/PowerQualityMonitor/_Structs/ST_PowerMonitor_InputField.TcDUT
TYPE ST_PowerMonitor_InputField EXTENDS st_PQVoltageData:
STRUCT
	r_loadshare					: 	REAL;
	ACQuality					:	ST_PQGridQualityData;
	Powerlock					: 	ARRAY [1..2] OF st_PQVoltageData;
END_STRUCT
END_TYPE

// ---- POUs/Objects/PowerQualityMonitor/_Structs/ST_PowerMonitor_OutputField.TcDUT
TYPE ST_PowerMonitor_OutputField EXTENDS st_PQVoltageData:
STRUCT
	r_loadshare					: 	REAL;
	ACQuality					:	ST_PQGridQualityData;
	Powerlock					: 	ARRAY [1..3] OF ST_PQPowerData;
END_STRUCT
END_TYPE

// ---- POUs/Objects/PowerStack/NetContactor/_Structs/ST_Netcontactor_service.TcDUT
TYPE ST_Netcontactor_service :
STRUCT
	Right			: ST_service_DigitalOutInWithSafety;
	Left			: ST_service_DigitalOutInWithSafety;
END_STRUCT
END_TYPE

// ---- POUs/Objects/PowerStack/_Structs/ST_Powermodule_Service.TcDUT
TYPE ST_Powermodule_Service :
STRUCT
	b_FieldBusControlEnable			: BOOL := TRUE;
	b_FanOn							: eForceBool;
END_STRUCT
END_TYPE

// ---- POUs/Objects/PowerStack/_Structs/ST_Powerstack_MaintenanceParams.TcDUT
TYPE ST_Powerstack_MaintenanceParams :
STRUCT
	ForceNetcontactor		: BOOL;
END_STRUCT
END_TYPE

// ---- POUs/Objects/PowerStack/_Structs/ST_Powerstack_Service.TcDUT
TYPE ST_Powerstack_Service :
STRUCT
	Netcontactor			: St_Netcontactor_service;
	PowermoduleMaster		: ST_Powermodule_Service;
	PowermoduleSlave		: ST_Powermodule_Service;
END_STRUCT
END_TYPE

// ---- POUs/Safety/ST_Safety_ContactorEDM.TcDUT
TYPE ST_Safety_ContactorEDM :
STRUCT
	b_MccbMasterEDM						: BOOL;
	b_MccbSlaveEDM						: BOOL;
	b_NetcontactorEDM					: BOOL;
	b_DcMccbEDM							: BOOL;
END_STRUCT
END_TYPE

// ---- POUs/Safety/ST_Safety_get.TcDUT
TYPE ST_Safety_get :
STRUCT
	b_SafetyOK					: BOOL;
	b_SafetyDcOK				: BOOL;
	b_EstopChannelAOK			: BOOL;		
	b_EstopChannelBOK			: BOOL;		
	b_InsulationMonitorOK		: BOOL;	
	b_MRCDBOK					: BOOL;	
	b_InverterDoorOK            : BOOL;
	b_ZptOK				        : BOOL;
END_STRUCT
END_TYPE

// ---- POUs/Safety/ST_Safety_ToSafetyPrg.TcDUT
TYPE ST_Safety_ToSafetyPrg :
STRUCT
	b_ErrorReset						: BOOL;
	b_EmergencyStopSoftwareOK			: BOOL;
	b_SafetyRunStop						: BOOL := TRUE;
	contactors							: ST_Safety_ContactorEDM;
END_STRUCT
END_TYPE

// ---- POUs/Objects/4Grouter/Struct/dwtoreal.TcDUT
TYPE dwtoreal :
UNION
	Registers	:	ARRAY[1..2] OF WORD;
	dwordvalue	:	dword;
	realvalue	:	REAL;
END_UNION
END_TYPE

// ---- POUs/Objects/4Grouter/Struct/eModemState.TcDUT
{attribute 'qualified_only'}
//{attribute 'strict'}
TYPE eModemState :
(
	Disconnected := 0,
	Connected := 1
);
END_TYPE

// ---- POUs/Objects/4Grouter/Struct/eNetworkState.TcDUT
{attribute 'qualified_only'}
//{attribute 'strict'}
TYPE eNetworkState :
(
	unknown := 0,
	searching := 1,
	Unregistered := 2,
	Registered := 3,
	Roaming := 4
	);
END_TYPE

// ---- POUs/Objects/4Grouter/Struct/eSimSelectionMode.TcDUT
{attribute 'qualified_only'}
{attribute 'strict'}
TYPE eSimSelectionMode :
(
	auto := 0,
	force_sim1 := 1,
	force_sim2 := 2
);
END_TYPE

// ---- POUs/Objects/4Grouter/Struct/eSimState.TcDUT
{attribute 'qualified_only'}
//{attribute 'strict'}
TYPE eSimState :
(
	no_sim := 0,
	Inserted := 1,
	active := 2,
	pin_fault := 3
);
END_TYPE

// ---- POUs/Objects/4Grouter/Struct/eSMSStatus.TcDUT
{attribute 'qualified_only'}
//{attribute 'strict'}
TYPE eSMSStatus :
(
	Idle 			:= 	0,
	NewMessage 		:= 	1,
	SendingMessage 	:= 	2,
	error			:=	3
);
END_TYPE

// ---- POUs/Objects/4Grouter/Struct/eWifiSecurityTypes.TcDUT
{attribute 'qualified_only'}
{attribute 'strict'}
{attribute 'to_string'}
TYPE eWifiSecurityTypes :
(
	none := 0,
	PSK2 := 1,
	SAE  := 2,
	SAE_mixed := 3,
	PSK := 4	
);
END_TYPE

// ---- POUs/Objects/4Grouter/Struct/eWifiStatus.TcDUT
{attribute 'qualified_only'}
TYPE eWifiStatus :
(
	invalid := 0,
	off := 1,
	searching := 2,
	Connected := 3,
	Starting := 4,
	Active := 5
);
END_TYPE

// ---- POUs/Objects/4Grouter/Struct/st_Device.TcDUT
TYPE st_Device :
STRUCT
	SystemUptime	:	UDINT;	
	Temperature		:	REAL;
	RouterSerial	:	STRING(32);
END_STRUCT
END_TYPE

// ---- POUs/Objects/4Grouter/Struct/st_GPS.TcDUT
TYPE st_GPS :
STRUCT
	Latitude 	: 	REAL;
	Longitude 	: 	REAL;
	FixTime 	: 	STRING(32);
	DateTime	:	DT;
	Speed		:	REAL;
	SatCount	:	UINT;
	Accuracy	:	REAL;	
END_STRUCT
END_TYPE

// ---- POUs/Objects/4Grouter/Struct/st_mobile.TcDUT
TYPE st_mobile :
STRUCT
	NetworkOperator				:	STRING(32);
	NetworkInfo					:	STRING(32);
	NetworkType					:	STRING(32);
	RSSI						:	DINT;
	ui_Sim1DataSendMonth		:	UINT;
	ui_Sim1DataReceivedMonth	:	UINT;
	ui_Sim2DataSendMonth		:	UINT;
	ui_Sim2DataReceivedMonth	:	UINT;
	s_EmergencySMSNumber		:	STRING(20);
	s_SecondarySMSNumber		:	STRING(20);
	s_EmergencySMSDevName		:	STRING(18);
	st_LatestSMSMessage			:	STRING(80);
	ModemState					:	eModemState;
	NetworkState				:	eNetworkState;
	ui_ActiveSim				:	UINT;
	SimStatus					:	eSimState;
END_STRUCT
END_TYPE

// ---- POUs/Objects/4Grouter/Struct/st_Router_Events.TcDUT
TYPE st_Router_Events :
STRUCT
	b_MBCommWarning		:	BOOL;
	b_NoSimWarning		:	BOOL;
	b_NoNetworkWarning	: 	BOOL;
	b_noGPSFixWarning	:	BOOL;
	b_SMSNotSendError	:	BOOL; 
	b_NoSMSNumberAvailable	:	BOOL;
	b_TimeUpdateFailed 	: BOOL;
END_STRUCT
END_TYPE

// ---- POUs/Objects/4Grouter/Struct/st_router_get.TcDUT
TYPE st_router_get :
STRUCT
	Device 		: 	st_Device;
	GPS			:	st_GPS;
	Mobile		:	st_mobile;
	Wifi		:	st_Wifi;
	e_SMSStatus : 	eSMSStatus;
	Events		:	st_Router_Events;
END_STRUCT
END_TYPE

// ---- POUs/Objects/4Grouter/Struct/ST_Router_params.TcDUT
TYPE ST_Router_params :
STRUCT
	IP_TELTONIKA		: STRING(16) := '192.168.1.1';
	MBPort_TELTONIKA 	: UINT := 502;
	T_MBTimeout			: TIME := T#2S;
	MinimumPhoneNumberLength	:UINT := 10;
	
	//temporary setup via stparams until integrated into HMI
	ManualSettings		:	st_router_set;
END_STRUCT
END_TYPE

// ---- POUs/Objects/4Grouter/Struct/ST_Router_set.TcDUT
TYPE ST_Router_set :
STRUCT
	EnableWifiClient	:	BOOL;
	WifiClientSSID		:	STRING(32) := 'MachineAccessPoint@VDL';
	WifiClientPass		:	STRING(32) := 'e4ff1c12kLL';
	WifiClientSecType	:	eWifiSecurityTypes := eWifiSecurityTypes.PSK2;
	
	EnableWifiAP		:	BOOL;
	WifiAPSSID			:	STRING(32) := 'ePU10_AP';
	WifiAPPass			:	STRING(32) := 'Welkom!VDL';
	WifiAPSecType		:	eWifiSecurityTypes := eWifiSecurityTypes.PSK2;
	
	SimSelectionMode	:	eSimSelectionMode := eSimSelectionMode.auto;
	Sim1Pin				:	STRING(4) := '0000';
	Sim2Pin				:	STRING(4) := '0000';
	
	UpdateSystemTime	:	BOOL;
	
	AutoRebootEnable	:	BOOL;
	ManualReboot		:	BOOL;
END_STRUCT
END_TYPE

// ---- POUs/Objects/4Grouter/Struct/st_Wifi.TcDUT
TYPE st_Wifi :
STRUCT
	WifiClienModeStatus		:	eWifiStatus;
	WifiAPModeStatus		:	eWifiStatus;
	WifiApNumberOfClients	:	Uint;
END_STRUCT
END_TYPE

// ---- POUs/Objects/ACDCCharger/Enums/eAcDcChargerState.TcDUT
{attribute 'qualified_only'}
{attribute 'strict'}
{attribute 'to_string'} 

TYPE eAcDcChargerState :
(
	init 		:= 0,
	off 		:= 1,
	Standby	 	:= 2,
	starting 	:= 4,
	running		:=	5,
	stopping	:=	6, 

	fault 		:= 7
);
END_TYPE

// ---- POUs/Objects/ACDCCharger/Structs/Hadi/E_ChargerState.TcDUT
TYPE E_ChargerState :
(
    Idle := 0,
    ModulesOff := 10,
    SetVI := 20,
    CheckVoltage := 30,
    EnableModules := 40,
    Running := 100,
    Shutdown := 200,
    OpenRelay := 210,
    Fault := 900
);
END_TYPE

// ---- POUs/Objects/ACDCCharger/Structs/Hadi/ST_CanId.TcDUT
TYPE ST_CanId :
STRUCT
    ExtendedBit : BOOL;   // Bit31 (should always be TRUE)
    ErrorCode   : BYTE;   // Bits 28..26
    DeviceNo    : BYTE;   // Bits 25..22
    CommandNo   : BYTE;   // Bits 21..16
    TargetAddr  : BYTE;   // Bits 15..8
    SourceAddr  : BYTE;   // Bits 7..0
END_STRUCT
END_TYPE

// ---- POUs/Objects/ACDCCharger/Structs/Hadi/ST_ChargerControl.TcDUT
TYPE ST_ChargerControl :
STRUCT
    (* Charger control *)
    bStartCharge      : BOOL;   // start charging sequence
    bStopCharge       : BOOL;   // stop charging sequence

    (* Module enable command *)
    bEnableModules    : BOOL;   // CMD 1A

    (* Setpoints *)
    rSetVoltage       : REAL;   // desired voltage [V]
    rSetCurrent       : REAL;   // desired current [A]

    (* Apply commands *)
    bApplyGroupSet    : BOOL;   // CMD 1B (group control)
    bApplyModuleSet   : BOOL;   // CMD 1C (module control)

    (* Target module *)
    ModuleTarget      : BYTE;   // module number (peer-to-peer)

    (* Hardware relay *)
    bSystemRelayCmd   : BOOL;   // command to close system relay
END_STRUCT
END_TYPE

// ---- POUs/Objects/ACDCCharger/Structs/Hadi/ST_Control.TcDUT
TYPE ST_Control :
STRUCT
	rLimitInputCurrent	: REAL;	// CMD 0F Limit input current on all power modules
//	stModuleControl		: ARRAY [0..10] OF REAL;
	bEnableDisable		: BOOL; // CMD 1A (Broadcastong or Group)
	rSetOutputVoltage	: REAL;	// CMD 1B
	rSetOutputCurrent	: REAL;	// CMD 1B
	bResetMode			: BOOL;	// CMD 1E
	
END_STRUCT
END_TYPE

// ---- POUs/Objects/ACDCCharger/Structs/Hadi/ST_Data.TcDUT
TYPE ST_Data :
STRUCT
	rSystemOutVoltageDc		: REAL;		// CMD 01
	rSystemOutCurrentDc		: REAL;		// CMD 01
	rNumberOfModules		: REAL;		// CMD 02
	stModuleData			: ARRAY [0..10] OF ST_ModuleData;
	
	
	
	
	
END_STRUCT
END_TYPE

// ---- POUs/Objects/ACDCCharger/Structs/Hadi/ST_ModuleControl.TcDUT
TYPE ST_ModuleControl :
STRUCT
	bEnableDisable		: BOOL; // CMD 1A
	rSetOutputVoltage	: REAL;	// CMD 1C
	rSetOutputCurrent	: REAL;	// CMD 1C
	
	
	
	
END_STRUCT
END_TYPE

// ---- POUs/Objects/ACDCCharger/Structs/Hadi/ST_ModuleData.TcDUT
TYPE ST_ModuleData :
STRUCT
	rOutVoltageDc		: REAL;	// CMD 03
	rOutCurrentDc		: REAL;	// CMD 03
	rTemprature			: REAL;	// CMD 04
	rStatus0			: REAL;	// CMD 04
	rStatus1			: REAL;	// CMD 04
	rStatus2			: REAL;	// CMD 04
	rVoltageL1L2		: REAL;	// CMD 06
	rVoltageL2L3		: REAL;	// CMD 06
	rVoltageL3L1		: REAL;	// CMD 06
	rExternalVoltageDc	: REAL;	// CMD 0C      this could be the same as rOutVoltageDc CMD 03
	ravilableCurrentDc	: REAL;	// CMD 0C
	
	 stStatus           : ST_ModuleStatus;  // decoded status bits
	 
	 bValid		: BOOL; // validate if data are updating
	
END_STRUCT
END_TYPE

// ---- POUs/Objects/ACDCCharger/Structs/Hadi/ST_ModuleStatus.TcDUT
TYPE ST_ModuleStatus :
STRUCT
	 (* STATUS 2 *)
    bPfcOff              : BOOL;	// Bit 7
    bInputOverVoltage    : BOOL;	// Bit 6	
    bInputUnderVoltage   : BOOL;	// Bit 5
    bInputAsymmetry      : BOOL;	// Bit 4
    bPhaseLost           : BOOL;	// Bit 3
    bLoadSharingError    : BOOL;	// Bit 2
    bModuleIdDuplicate   : BOOL;	// Bit 1
    bPowerLimitation     : BOOL;	// Bit 0

    (* STATUS 1 *)
    bCanTimeout          : BOOL;	// Bit 7    /////////
    bSlowStartup         : BOOL;	// Bit 6
    bOutputOverVoltage   : BOOL;	// Bit 5
    bTempHigh            : BOOL;	// Bit 4
    bFanError            : BOOL;	// Bit 3
    bModuleProtection    : BOOL;	// Bit 2
    bModuleError         : BOOL;	// Bit 1      ////////////
    bDcSideOff           : BOOL;	// Bit 0

    (* STATUS 0 *)
    bDischargeAbnormal   : BOOL;	// Bit 5
    bMpptSwitchMode      : BOOL;	// Bit 4
    bPfcAbnormal         : BOOL;	// Bit 3
    bInternalCommError   : BOOL;	// Bit 2
    bOutputShortCircuit  : BOOL;	// Bit 0
END_STRUCT
END_TYPE

// ---- POUs/Objects/ACDCCharger/Structs/ST_ACDCCharger_events.TcDUT
TYPE ST_ACDCCharger_events :
STRUCT
	b_CommunicationFault			:	BOOL;
	b_BuscouplerNotFound			:	BOOL;
	b_ACUnderVoltageDeratingActive	: 	BOOL;
	b_BatteryLimitDeratingActive	:	BOOL;
	b_TemperatureDeratingActive		:	BOOL;
	b_CurrentLimitActive			:	BOOL;
	b_SOCLimitReached				:	BOOL;
	b_FailedToGenerateDCOutput		:	BOOL;
	B_ACPhaselossFault				:	BOOL;
	B_ACUndervoltage				:	BOOL;
	B_ACOvervoltage					:	BOOL;
END_STRUCT
END_TYPE

// ---- POUs/Objects/ACDCCharger/Structs/ST_ACDCCharger_get.TcDUT
TYPE ST_ACDCCharger_get :
STRUCT
	e_SystemStatus			: eAcDCChargerState := eACDCChargerState.init;
	
	by_NoModulesActive		: BYTE;	
	by_NoModulesInstalled	: BYTE;
	e_ChargerStatus 		: ARRAY [0..6] OF eAcDcChargerState;
	
	ar_ACvoltage			: ARRAY [0..3] OF REAL;
	r_AvailablePower		: REAL;
	ACmeasurements			: ST_PQPowerData;
	r_DcVoltage	   			: REAL;
	r_DcCurrent				: REAL;
	r_DcPower				: REAL;

	Events					: ST_ACDCCharger_events;	

END_STRUCT
END_TYPE

// ---- POUs/Objects/ACDCCharger/Structs/ST_ACDCCharger_params.TcDUT
TYPE ST_ACDCCharger_params :
STRUCT
	b_ACDCChargerFitted		:	BOOL;
	ui_NrOfInstalledModules	:	UINT	:=	2;
	ui_ModuleDesignPower	:	Uint	:=	30;
	r_VoltageWindow			:	REAL	:=  2;
	GridVoltageHysteresis	: 	REAL	:=	2;
	BMSChargeLimitRampRate	:	REAL	:=	0.5; //DC amps per cycle;
	SocHysteresis			:	Real	:=	2;
END_STRUCT
END_TYPE

// ---- POUs/Objects/ACDCCharger/Structs/ST_ACDCCharger_set.TcDUT
TYPE ST_ACDCCharger_set :
STRUCT
	b_enable			: 	BOOL;
	e_ControlType		: 	ePowerControlType;
	r_currentSetpoint 	: 	REAL;
	r_powersetpoint		: 	REAL;
	r_MinGridVoltage	:	REAL;
	r_SocTarget			:	REAL;
END_STRUCT
END_TYPE

// ---- POUs/Objects/ACDCCharger/Structs/ST_SystemDiagnostic.TcDUT
TYPE ST_SystemDiagnostic :
STRUCT

    (* ===== GLOBAL STATUS ===== *)
    bAnyError          : BOOL;
    bAnyWarning        : BOOL;

    (* ===== ERRORS (CRITICAL) ===== *)
    bError_OutputOV    : BOOL;
    bError_OverTemp    : BOOL;
    bError_ShortCircuit: BOOL;
    bError_ModuleError : BOOL;
    bError_CommLost    : BOOL;
    bError_PhaseLost   : BOOL;

    (* ===== WARNINGS ===== *)
    bWarn_InputOV      : BOOL;
    bWarn_InputUV      : BOOL;
    bWarn_FanError     : BOOL;
    bWarn_PowerLimit   : BOOL;
    bWarn_TempHigh     : BOOL;
    bWarn_CurrentLimit : BOOL;

    (* ===== SYSTEM INFO ===== *)
    bAllModulesOff     : BOOL;
    bAllModulesOn      : BOOL;

END_STRUCT
END_TYPE

// ---- POUs/Objects/ACDCCharger/Structs/ST_SystemEval.TcDUT
TYPE ST_SystemEval :
STRUCT
    bAllModulesOff : BOOL;
    bAnyModuleActive : BOOL;
    bAnyModuleFault : BOOL;
    bGridOk : BOOL;

    rTotalAvailableCurrent : REAL;
    rMaxTemperature : REAL;
    iHealthyModules : INT;
END_STRUCT
END_TYPE

// ---- POUs/Objects/Enclosure/Climate/ST_Enclosureclimate_events.TcDUT
TYPE ST_Enclosureclimate_events :
STRUCT
	b_HumidityHigh 			: BOOL;
	b_HumidityTooHigh 		: BOOL;
	b_TemperatureHigh		: BOOL;
	b_TemperatureTooHigh	: BOOL;
	b_TemperatureLow		: BOOL;
	b_TemperatureTooLow		: BOOL;
	b_AIOverrange			: BOOL;
	b_AIUnderrange			: BOOL;
	b_AIError				: BOOL;
	b_DewpointTooHigh		: BOOL;
END_STRUCT
END_TYPE

// ---- POUs/Objects/Enclosure/Climate/ST_EnclosureClimate_get.TcDUT
TYPE ST_EnclosureClimate_get :
STRUCT
	r_Humidity			: REAL;
	r_Temperature		: REAL;
	r_Dewpoint			: REAL;
	events				: ST_EnclosureClimate_events;
END_STRUCT
END_TYPE

// ---- POUs/Objects/Enclosure/Climate/ST_EnclosureClimate_Params.TcDUT
TYPE ST_EnclosureClimate_Params :
STRUCT
	r_HumidityHysteris		: REAL:= 2;
	r_HumidityHigh			: REAL:= 80;
	r_HumidityTooHigh		: REAL:= 90;
	r_TemperatureHysteris	: REAL:= 2;
	r_TemperatureHigh		: REAL:= 40;
	r_TemperatureTooHigh	: REAL:= 50;
	r_TemperatureLow		: REAL:= -10;
	r_TemperatureTooLow		: REAL:= -20;
	
	r_EnclosureConditioningTempMin					: REAL := 10.0;
	r_EnclosureConditioningTempMax					: REAL := 40.0;
END_STRUCT
END_TYPE

// ---- POUs/Objects/Enclosure/Doors/ST_DoorsNLocks_get.TcDUT
TYPE ST_DoorsNLocks_get :
STRUCT
	b_BuscouplerOK					: Bool;
	b_ClientpanelDoorOpen			: BOOL;
	b_ControlPanelDoorOpen			: BOOL;	
	b_InverterDoorOpen				: BOOL;
	b_UPSBatteryDoorOpen			: BOOL;
	b_MainBatteryLeftDoorOpen		: BOOL;
	b_MainBatteryRightDoorOpen		: BOOL;
END_STRUCT
END_TYPE

// ---- POUs/Objects/Enclosure/LedIndicator/BeckhoffController/eDCstate.TcDUT
{attribute 'qualified_only'}
{attribute 'strict'}
TYPE eDCstate :
(
	charging :=-1,
	idle := 0,
	discharging := 1
);
END_TYPE

// ---- POUs/Objects/Enclosure/LedIndicator/BeckhoffController/eLEDSteps.TcDUT
{attribute 'qualified_only'}
{attribute 'strict'}
TYPE eLEDSteps :
(
	initialise,	
	running
);
END_TYPE

// ---- POUs/Objects/Enclosure/LedIndicator/BeckhoffController/eSystemStatus.TcDUT
{attribute 'qualified_only'}
{attribute 'strict'}
TYPE eSystemStatus :
(
	off			:= 0,	// off
	neutral 	:= 1, 	(*white*)
	normal		:= 2, 	// green
	attention	:= 3,	// blue 100charge 0discharge
	warning		:= 4,	// yellow
	error		:= 5	// red	
) BYTE;
END_TYPE

// ---- POUs/Objects/Enclosure/LedIndicator/BeckhoffController/LEDColor.TcDUT
TYPE LEDColor :
STRUCT	
	red 	:USINT;
	green	:USINT;
	blue	:USINT;
	white	:USINT;
END_STRUCT
END_TYPE

// ---- POUs/Objects/Enclosure/LedIndicator/BeckhoffController/LEDCommands.TcDUT
TYPE LEDCommands :
STRUCT
	
	fill 		: USINT := 1;
	clear 		: USINT	:= 2;
	copy 		: USINT	:= 3;
	movePixel 	: USINT	:= 4;
	reverse 	: USINT	:= 7;
END_STRUCT
END_TYPE

// ---- POUs/Objects/Enclosure/LedIndicator/BeckhoffController/LEDControl.TcDUT
TYPE LEDControl :
STRUCT
	execute 	: BIT;
	send		: BIT;
	update		: BIT;
	command		: USINT;(*LEDCommands*)
	index 		: UINT;
	length		: UINT;
	parameter	: UINT;
	color 		: LEDColor;
END_STRUCT
END_TYPE

// ---- POUs/Objects/Enclosure/LedIndicator/BeckhoffController/LEDStatus.TcDUT
TYPE LEDStatus :
STRUCT
	busy				: BIT;
	transmit			: BIT;
	sendAcknowledge 	: BIT;
	updateAcknowledge	: BIT;
	commandAcknowledge	: BIT;
	commandReject		: BIT;
	warning				: BIT;
	error				: BIT;
	InputCycleCounter	: USINT;
END_STRUCT
END_TYPE

// ---- POUs/Objects/Enclosure/LedIndicator/eColorOrder.TcDUT
{attribute 'qualified_only'}

TYPE eColorOrder :
(
	RGB := 0,
	GRB := 1
);
END_TYPE

// ---- POUs/Objects/Enclosure/LedIndicator/ST_Ledstrip_get.TcDUT
TYPE ST_Ledstrip_get :
STRUCT
	b_error		: BOOL;
	BeckhoffLed	: BOOL;
END_STRUCT
END_TYPE

// ---- POUs/Objects/Enclosure/LedIndicator/st_Ledstrip_MachineData.TcDUT
TYPE st_Ledstrip_MachineData :
STRUCT
	r_SOC 					: REAL;
	r_DCCurrent				: REAL;
	e_systemStatus 			: eSystemStatus;
END_STRUCT
END_TYPE

// ---- POUs/Objects/Enclosure/LedIndicator/st_Ledstrip_params.TcDUT
TYPE st_Ledstrip_params :
STRUCT
	IP				: STRING 	:= '192.168.1.43'; //arduino controller only
	Numleds			: BYTE		:= 116;
	ColorOrder		: eColorOrder := eColorOrder.GRB;
END_STRUCT
END_TYPE

// ---- POUs/Objects/Enclosure/_struct/ST_Enclosure_get.TcDUT
TYPE ST_Enclosure_get :
STRUCT
	climate				: ST_EnclosureClimate_Get;
	doors				: ST_DoorsNLocks_get;
	ledstrip			: ST_Ledstrip_get;
END_STRUCT
END_TYPE

// ---- POUs/Objects/Enclosure/_struct/st_Enclosure_params.TcDUT
TYPE st_Enclosure_params :
STRUCT
	climate			: ST_EnclosureClimate_params;
	ledstrip		: st_Ledstrip_params;
END_STRUCT
END_TYPE

// ---- POUs/Objects/Enclosure/_struct/ST_enclosure_set.TcDUT
TYPE ST_enclosure_set :
STRUCT
	by_LedBrightness 	: BYTE := 100;
END_STRUCT
END_TYPE

// ---- POUs/Objects/GenComm/eNums/eGenControlProtocol.TcDUT
{attribute 'qualified_only'}
{attribute 'strict'}
TYPE eGenControlProtocol :
(
	None := 0,
	AGC150 := 1
);
END_TYPE

// ---- POUs/Objects/GenComm/eNums/eGenOperationMode.TcDUT
{attribute 'qualified_only'}
{attribute 'strict'}
TYPE eGenOperationMode :
(
	None := 0,
	BlockMode := 1,
	ManualMode := 2,
	SemiAuto := 3,
	Auto	:=	4,
	Test	:=	5
);
END_TYPE

// ---- POUs/Objects/GenComm/eNums/eOnOffState.TcDUT
{attribute 'qualified_only'}
{attribute 'strict'}
TYPE eOnOffState :
(
	none := 0,
	Enable := 1,
	Disable := 2
);
END_TYPE

// ---- POUs/Objects/GenComm/Structs/ST_AGC150_Set.TcDUT
TYPE ST_AGC150_Set :
STRUCT
	IP					:	STRING	:=	'192.168.2.21';
	DroopEnable			: 	BOOL;
	GenOn				:	eOnOffState := eOnOffState.none;
	GenBreakerOn		:	eOnOffState := eOnOffState.none;	
	MainBreakerON		:	eOnOffState := eOnOffState.none;
	GenAutoSyncOn		:	eOnOffState := eOnOffState.none;
	OperationMode		:	eGenOperationMode := eGenOperationMode.Auto;
	AutoStartStop		:	BOOL;
	
	bIslandModeEnable		:	BOOL;
	bAMFModeEnable			:	BOOL;
	bPeakshavingEnable		: 	BOOL;
	bFixedPowerEnable		:	BOOL := TRUE;
	bMPE					:	BOOL;

	Pset			:	REAL;	//0..100%
	Qset			:	REAL;	//60..100 = 0.6..1
	PFset			:	REAL := 1;	//-100..100%
	FreqRegulator	:	REAL; 	//-100..100 = -10..+10% of nominal
	VoltRegulator	:	REAL; 	//-100..100 = -10..+10% of nominal
	U_Fdroopset		: 	REAL := 4; 	//0..100 = 0..+10% of nominal
END_STRUCT
END_TYPE

// ---- POUs/Objects/GenComm/Structs/ST_GenComm_Params.TcDUT
TYPE ST_GenComm_Params :
STRUCT
	IP					:	STRING	:=	'192.168.2.21';
	GenControlProtocol	: 	eGenControlProtocol := eGenControlProtocol.None;
END_STRUCT
END_TYPE

// ---- POUs/Objects/GenComm/Structs/ST_Genset_Get.TcDUT
TYPE ST_Genset_Get :
STRUCT
	CommunicationOK		: 	BOOL;
	FuelLow				: 	BOOL;
	FuelCritical		: 	BOOL;
		
	bGenBreakerClosed	:	BOOL;
	bMainBreakerClosed	:	BOOL;
	bGenRunning			:	BOOL;
	bGenVoltFreqOK		:	BOOL;
	bMainsFailure		:	BOOL;
	
	eActiveGenMode		:	eGenOperationMode;
	bIslandModeActive	:	BOOL;
	bAMFActive			:	BOOL;
	bPeakshaveActive	:	BOOL;
	bFixedPowerActive	:	BOOL;

	ar_LineVoltage	:	ARRAY[0..3] OF REAL;
	ar_PhaseVoltage	:	ARRAY[0..3] OF REAL;
	ar_Frequency	:	ARRAY[0..3] OF REAL;
	ar_Current		:	ARRAY[0..3] OF REAL;
	ar_PowerFactor	: 	ARRAY[0..0] OF REAL;
	ar_ActivePower 	:   ARRAY[0..3] OF REAL;
	ar_ReactivePower: 	ARRAY[0..0] OF REAL;
	ar_ApparentPower:	ARRAY[0..0] OF REAL;
	
	
END_STRUCT
END_TYPE

// ---- POUs/Objects/GenComm/Structs/ST_Genset_Set.TcDUT
TYPE ST_Genset_Set :
STRUCT
	enable			:  	BOOL;
	StartStop		:	BOOL; //true = start;
	Pset			:	REAL;	//0..100%
	Qset			:	REAL;	//60..100 = 0.6..1
	PFset			:	REAL;	//0 - 1;
	Uset			: 	REAL;
	Fset			: 	REAL;
	U_Fdroopset		: 	REAL := 4;
	GensetMode		: 	eGensetMode := eGensetMode.FixedPower;
END_STRUCT
END_TYPE

// ---- POUs/Objects/HartingIO/ST_HartingIO_get.TcDUT
TYPE ST_HartingIO_get :
STRUCT
	b_DigitalInput1Active		:	BOOL;
	b_DigitalInput2Active		:	BOOL;
	b_GenLowFuel				:	BOOL;
	b_ExtSystemShutdownRequest	:	BOOL;
	b_ExtEMstopOK				: 	BOOL;
	b_ExtEMstopActive			: 	BOOL;
END_STRUCT
END_TYPE

// ---- POUs/Objects/HartingIO/ST_HartingIO_params.TcDUT
TYPE ST_HartingIO_params :
STRUCT
	PrimaryOutputContactSignal		: 	eOutputContactSignal := eOutputContactSignal.GenStartStop;
	SecondaryOutputContactSignal	:	eOutputContactSignal := eOutputContactSignal.None;
	PrimaryInputContactSignal		: 	eInputSignal := eInputSignal.None;
	SecondaryInputContactSignal		: 	eInputSignal := eInputSignal.None;
	AO1Target				: eAOTarget := eAOTarget.Genset;
	AO2Target				: eAOTarget	:= eAOTarget.hPU;
END_STRUCT
END_TYPE

// ---- POUs/Objects/HartingIO/ST_HartingIO_set.TcDUT
TYPE ST_HartingIO_set :
STRUCT
	w_SwitchControlSignals		: 	WORD; // control signals for output contact
	r_manualAnalogOutput		: 	REAL; // 0 - 100%
	r_gensetAnalogOutput		: 	REAL; // 0 - 100%
	r_HpuAnalogOutput			: 	REAL; // 0 - 100%
END_STRUCT
END_TYPE

// ---- POUs/Objects/HartingIO/_Enum/eAOTarget.TcDUT
{attribute 'qualified_only'}
{attribute 'strict'}
TYPE eAOTarget:
(
	manual 	:= 0,
	Genset	:= 1,
	hPU		:= 2
);
END_TYPE

// ---- POUs/Objects/HartingIO/_Enum/eInputSignal.TcDUT
{attribute 'qualified_only'}

TYPE eInputSignal :
(
	None 			:= 	0,
	GenLowFuel 		:= 	1,
	StopOperation 	:= 	2,
	EMstop			:=	3
) UINT;
END_TYPE

// ---- POUs/Objects/HartingIO/_Enum/eOutputContactSignal.TcDUT
{attribute 'qualified_only'}

TYPE eOutputContactSignal :
(
	None 			:= 	0,
	FireAlarm 		:= 	1,
	GenStartStop 	:= 	2,
	HPU				:= 	3,
	SystemActive	:=	4,
	PVenable		:= 	5,
	ManualOpen		:=	99,
	ManualClose		:=	100
) UINT;
END_TYPE

// ---- POUs/Objects/InterMachineCom/ST_InterMachineCom_Master.TcDUT
TYPE ST_InterMachineCom_Master :
STRUCT
	PS		: REAL; //Power setpoint, scale 0.1% 
	QS		: REAL; // Reactive Setpoint, scale 0.1%
	CW		: WORD; // ControlWord, b0: Start, b1: Stop, b2: shutdown, b3: EMstop, b4: Reset, b15: watchdog signal
END_STRUCT
END_TYPE

// ---- POUs/Objects/InterMachineCom/ST_IntermachineCom_params.TcDUT
TYPE ST_IntermachineCom_params :
STRUCT
	InternalBrokerIP		: STRING := '10.4.0.41';
	MasterPublishRate		: TIME := T#20MS;
	SlavePublishRate		: TIME := T#1S;
	WatchdogPulseRate		: TIME := T#2S;
	EMstopCoupling			: BOOL;
END_STRUCT
END_TYPE

// ---- POUs/Objects/InterMachineCom/st_InterMachineCom_Slave.TcDUT
TYPE st_InterMachineCom_Slave :
STRUCT
	ACP : UINT; //available charge power [kW]
	ADP	: UINT; //available discharge power [kW]
	AQ	: UINT; //available Reactive Power [kvar]
	SW	: WORD; //status word: b0: standby, b1: running, b2: Stopped, b3: Discharge Only, b4: Charge Only, b5: warning active, b6: Alarm active, b7: EMstop active, b15: watchdogbit
END_STRUCT
END_TYPE

// ---- POUs/Objects/InterMachineCom/ST_InterMachineCom_SlaveConData.TcDUT
TYPE ST_InterMachineCom_SlaveConData :
STRUCT
	enable			: BOOL;
	BrokerIP		: STRING;
END_STRUCT
END_TYPE

// ---- POUs/Objects/InternalPowerSupply/eNums/e400VSupplySource.TcDUT
{attribute 'qualified_only'}
{attribute 'strict'}
{attribute 'to_string'}

TYPE e400VSupplySource :
(
	none := 0,
	grid := 1,
	CEE := 2
);
END_TYPE

// ---- POUs/Objects/InternalPowerSupply/eNums/eSupplyState.TcDUT
{attribute 'qualified_only'}
{attribute 'strict'}
TYPE eSupplyState :
(
	enum_member := 0
);
END_TYPE

// ---- POUs/Objects/InternalPowerSupply/Structs/ST_InternalPowerStatus.TcDUT
TYPE ST_InternalPowerStatus :
STRUCT
	b_Status_24VDC		:	BOOL;
	b_Status_HVDC		:	BOOL;
	b_Status_400VAC		:	BOOL;
END_STRUCT
END_TYPE

// ---- POUs/Objects/InternalPowerSupply/Structs/ST_InternalPowerSupply_Events.TcDUT
TYPE ST_InternalPowerSupply_Events :
STRUCT
	b_DCPSUFault				: 	BOOL; //fuse blown or psu_ok signal lost
	b_ACPSUFault				: 	BOOL;
	b_GridInputFuseTripped		:	BOOL;
	b_HVDCShutdownTimeExceeded	:	BOOL;
	b_UPSLowShutdown			:	BOOL;	//System shutdown event when ups battery drains during operation
	b_CEEPreventsShutdown		:	Bool;
END_STRUCT
END_TYPE

// ---- POUs/Objects/InternalPowerSupply/Structs/ST_InternalPowerSupply_Get.TcDUT
TYPE ST_InternalPowerSupply_Get :
STRUCT
	CEEInputActive		:	BOOL;
	b_24VdcAvailable	:	BOOL;
	b_HVDCAvailable		:	BOOL;
	b_400VACAvailable	:	BOOL;	
	
	UPS					:	REFERENCE TO ST_UPSGet;	
	Events				:	st_InternalPowerSupply_Events;
END_STRUCT
END_TYPE

// ---- POUs/Objects/InternalPowerSupply/Structs/ST_InternalPowerSupply_Params.TcDUT
TYPE ST_InternalPowerSupply_Params :
STRUCT
	i_ACStartupDelay : INT := 100; //ms
	i_DCPSU_StartupDelay: INT := 1000; //ms
	i_ACPSU_StartupDelay: INT := 1000; //ms
	
	//trigger level before Battery low error is issued. 
	usi_UPSBattLowErrorSOC		:	USINT 	:= 30;
	//UPS charging request was apparently denied. System should shutdown? 
	usi_UPSBattLowwarningSOC	:	USINT 	:= 50;
	//trigger level before Battery low warning is issued and UPS charging is requested from Internal power supply
	LowBatteryShutdownTimer		:	TIME := T#10M;
	
	//Battery self test interval (days). 0 means disable
	t_UPSBattSelfTestInterval	:	TIME := T#30D;
	
END_STRUCT
END_TYPE

// ---- POUs/Objects/InternalPowerSupply/Structs/ST_InternalPowerSupply_PowerDemand.TcDUT
TYPE ST_InternalPowerSupply_PowerDemand :
STRUCT
	b_Demand_24V	:	BOOL;
	b_Demand_400V	:	BOOL;
	b_Demand_HVDC	:	BOOL;
END_STRUCT
END_TYPE

// ---- POUs/Objects/InternalPowerSupply/UPS/eNums/eUPSState.TcDUT
{attribute 'qualified_only'}
{attribute 'strict'}
TYPE eUPSState :
(
	Inoperative 	:= 0,
	Input_Active	:= 1,
	On_Battery		:= 2
);
END_TYPE

// ---- POUs/Objects/InternalPowerSupply/UPS/Structs/ST_UPSData.TcDUT
TYPE ST_UPSData :
STRUCT
	udi_StatusFunctions 		: 	UDINT;
	udi_StatusInterface 		: 	UDINT;
	ui_InputVoltage				:	UINT;
	ui_InputCurrent				:	UINT;
	ui_OutputVoltage			:	UINT;
	ui_OutputCurrent			:	UINT;
	ui_BatteryVoltage			: 	UINT;
	ui_BatteryChargingCurrent 	: 	UINT;
	ui_BatteryTemperature 		: 	UINT;
	ui_DeviceTemperature		: 	UINT;
	udi_SOC 					:	UDINT;
	ui_TuPCShutdown				:	UINT;
	ui_SOH						:	UINT;
END_STRUCT
END_TYPE

// ---- POUs/Objects/InternalPowerSupply/UPS/Structs/ST_UPSEvents.TcDUT
TYPE ST_UPSEvents :
STRUCT
	b_BatteryLowInfo		:	BOOL;	//initialize DC conditioning
	b_BatteryLowWarning		:	BOOL;	//Battery charging failed, consider shutdown
	b_BatteryLowError		:	BOOL;	//Battery level critical, System should shutdown
	b_NoBatteryError		:	BOOL;	//no Battery voltage detected?
	b_InputVoltageWarning	:	BOOL;	//ipsstate says 24v is available, but no input is seen.
	
	b_UPSBatteryCalibrationActive	:	Bool;
END_STRUCT
END_TYPE

// ---- POUs/Objects/InternalPowerSupply/UPS/Structs/ST_UPSGET.TcDUT
TYPE ST_UPSGET :
STRUCT
	r_InputVoltage			:	REAL;
	r_OutputVoltage			:	REAL;
	r_BatteryVoltage		:	REAL;
	r_OutputCurrent			: 	REAL;
	ui_SOC					:	UINT	:=	100;
	
	b_ChargerActive			:	BOOL;
	b_SystemOnBattery		:	BOOL;
	b_SystemOnDCInput		:	BOOL;
	
	ui_UPSBatteryHealth		:	uint := 99;
	
	Events			:	ST_UPSEvents;
END_STRUCT
END_TYPE

// ---- POUs/Objects/NeutralTransformer/_Struct/ST_NeutralTransformer_events.TcDUT
TYPE ST_NeutralTransformer_events :
STRUCT
	b_TemperatureHighPhase						: ARRAY [1..3] OF BOOL; //1=L1, 2=L2, 3=L3
	b_TemperatureTooHighPhase					: ARRAY [1..3] OF BOOL; //1=L1, 2=L2, 3=L3
	b_VoltageUnbalanceHigh										: BOOL;
	b_VoltageUnbalanceTooHigh									: BOOL;
	b_NeutralCurrentHigh										: BOOL;
	b_NeutralCurrentTooHigh										: BOOL;
	
END_STRUCT
END_TYPE

// ---- POUs/Objects/NeutralTransformer/_Struct/ST_NeutralTransformer_Get.TcDUT
TYPE ST_NeutralTransformer_Get :
STRUCT
	b_active									: BOOL;
	r_TemperaturePhase							: ARRAY [0..6] OF REAL;
	r_Powerload									: REAL;
	r_ratedPower								: REAL; //kva
	events										: ST_NeutralTransformer_events;
END_STRUCT
END_TYPE

// ---- POUs/Objects/NeutralTransformer/_Struct/ST_Neutraltransformer_params.TcDUT
TYPE ST_Neutraltransformer_params :
STRUCT
	ui_ratedpower					: UINT := 60; // kVA
	by_TemperatureHighWarning		: BYTE := 80;
	by_TemperatureHighAlarm			: BYTE := 90;
	ui_TemperatureHighTripDelay		: UINT := 10; // seconds
	by_VoltageUnbalanceWarning		: BYTE := 10; // %
	by_VoltageUnbalanceAlarm		: BYTE := 20; // %
	ui_VoltageUnbalanceTripDelay	: UINT := 10;// seconds
	r_OCTripFactor					: REAL := 1.4;  //Overcurrent trip factor software
END_STRUCT
END_TYPE

// ---- POUs/Objects/PeakshaveBox/DUTs/ePSBMode.TcDUT
{attribute 'qualified_only'}
{attribute 'strict'}
{attribute 'to_string'}
TYPE ePSBMode :
(
	None 				:= 0,
	Monitor				:= 1,
	MonitorControl		:= 2	
);
END_TYPE

// ---- POUs/Objects/PeakshaveBox/ST_PeakShaveBox_Get.TcDUT
TYPE ST_PeakShaveBox_Get :
STRUCT
	PSBmode				: ePSBMode;
	Powermonitor 		: st_PQVoltageData;
	PowerQuality		: St_PQGridQualityData;
	PowerStatus			: ST_PQstatusData;
	r_MaxCTCurrent		: REAL:= 4000;
	b_buscouplerReady	: BOOL;
	b_active			: BOOL;
	b_dataOK			: BOOL;
	b_ContactorFb		: BOOL;
	b_SyncFb			: BOOL;
	b_SettingsChangePending	:	BOOL;
END_STRUCT
END_TYPE

// ---- POUs/Objects/PeakshaveBox/ST_peakshavebox_params.TcDUT
TYPE ST_peakshavebox_params :
STRUCT
	ExtBreakerControl	: BOOL := FALSE; 
END_STRUCT
END_TYPE

// ---- POUs/Objects/PeakshaveBox/ST_PeakshaveBox_Set.TcDUT
TYPE ST_PeakshaveBox_Set :
STRUCT
	b_ContactorClose : BOOL;
	b_BreakerControl : BOOL;
	ui_CtRange		 : UINT := 1000;
	r_VtPrimair		 : REAL;
	r_VtSecundair	 : REAL;	 
	b_InverseCTdirection: BOOL;
END_STRUCT
END_TYPE

// ---- POUs/Objects/PLCStatus/Enum/eFTPState.TcDUT
{attribute 'qualified_only'}
{attribute 'strict'}
{attribute 'to_string'}
TYPE
	eFTPState :(
		Disconnected := 0,	
		Connecting := 1,      
		Downloading := 2,      
		Success := 3,    
		Failure := 4
	);
END_TYPE

// ---- POUs/Objects/PLCStatus/Enum/eInstalState.TcDUT
{attribute 'qualified_only'}
{attribute 'strict'}
TYPE eInstalState :
(
	InProgress := 0,
	Success	   := 1,
	Failure	   := 2
);
END_TYPE

// ---- POUs/Objects/PLCStatus/Enum/eNetcomState.TcDUT
{attribute 'qualified_only'}
{attribute 'strict'}
{attribute 'To_string'}
TYPE eNetcomState :
(
	NotConnected := 0,
	OK:=1,
	Warning:=2,
	Error:=3
);
END_TYPE

// ---- POUs/Objects/PLCStatus/ST_EL9410.TcDUT
TYPE ST_EL9410 :
STRUCT
	bit_UpUndervoltage	: BIT;
	bit_UsUndervoltage	: BIT;
	ui_state			: UINT;
END_STRUCT
END_TYPE

// ---- POUs/Objects/PLCStatus/ST_PLCstate_get.TcDUT
TYPE ST_PLCstate_get :
STRUCT
	r_CPUload		: REAL;
	e_ProfinetState	: eNetcomState;
	e_EthercatState	: eNetcomState;
END_STRUCT
END_TYPE

// ---- POUs/Objects/PLCStatus/ST_PLC_events.TcDUT
TYPE ST_PLC_events :
STRUCT
	b_EthercatMasterFault		: BOOL;
END_STRUCT
END_TYPE

// ---- POUs/Objects/PowerStack/NetContactor/eNetcontMode.TcDUT
{attribute 'qualified_only'}
{attribute 'strict'}
TYPE eNetcontMode :
(
	auto := 0,
	left := 1,
	right := 2,
	none := 3
);
END_TYPE

// ---- POUs/Objects/PowerStack/NetContactor/_Structs/ST_Netcontactor_Events.TcDUT
TYPE ST_Netcontactor_Events :
STRUCT
	b_AMFEnabled							: BOOL;
	b_ContactorRightFbFault					: BOOL;
	b_ContactorLeftFbFault					: BOOL;
	b_ContactorFbTimeout					: BOOL;
	b_PhaseRotationFault					: BOOL;
	b_IllegalLeftFieldSelected				: BOOL;
END_STRUCT
END_TYPE

// ---- POUs/Objects/PowerStack/NetContactor/_Structs/ST_Netcontactor_get.TcDUT
TYPE ST_Netcontactor_get :
STRUCT
	e_NetConState					: eNetcontactorState;
	b_SyncCloseCommand				: BOOL;
	b_NetConFb						: BOOL;
	b_NetcontRightFb				: BOOL;
	b_NetcontLeftFb					: BOOL;
	events							: ST_Netcontactor_events;
END_STRUCT
END_TYPE

// ---- POUs/Objects/PowerStack/NetContactor/_Structs/ST_Netcontactor_set.TcDUT
TYPE ST_Netcontactor_set :
STRUCT
	e_ACRotationState				: eACRotationState; // 0:No AC, 1: AC CLOCKWISE, 2: AC ANTI-CLOCKWISE
	e_ClosingRequest				: eNetcontMode;
	b_ACdetected					: BOOL;
	b_RotationSwitchEnable			: BOOL;
	b_SynchronizedToD7				: BOOL;
END_STRUCT
END_TYPE

// ---- POUs/Objects/PowerStack/_Enums/eInverterModes.TcDUT
{attribute 'qualified_only'}
{attribute 'strict'}
{attribute 'to_string'}
TYPE eInverterModes :
(
	Afe := 0,
	Island := 1,
	Microgrid := 2
);
END_TYPE

// ---- POUs/Objects/PowerStack/_Enums/eNetContactorState.TcDUT
{attribute 'qualified_only'}
{attribute 'strict'}
{attribute 'to_string'}
TYPE eNetContactorState :
(
	Open 			:= 0,
	RightClosed		:= 1,
	LeftClosed		:= 2
);
END_TYPE

// ---- POUs/Objects/PowerStack/_Enums/ePLM.TcDUT
{attribute 'qualified_only'}
{attribute 'strict'}
{attribute 'to_string'}

TYPE ePLM: //power limiting 
(
	FreqShift := 0,
	VoltShift := 1,
	FreqVoltShift := 2,
	Shutdown := 3
);
END_TYPE

// ---- POUs/Objects/PowerStack/_Enums/ePowerModes.TcDUT
{attribute 'qualified_only'}
{attribute 'strict'}
{attribute 'to_string'}
TYPE ePowerModes :
(
	DroopZeroStart 		:= 0,
	Droop				:= 1,
	Isochronous			:= 2
);
END_TYPE

// ---- POUs/Objects/PowerStack/_Enums/ePowerModuleThrottlingState.TcDUT
{attribute 'qualified_only'}
{attribute 'strict'}
TYPE ePowerModuleThrottlingState :
(
	None := 0,
	FilterTemp := 1,
	InverterTemp:= 2,
	Overvoltage := 3
);
END_TYPE

// ---- POUs/Objects/PowerStack/_Enums/ePowerstate.TcDUT
{attribute 'qualified_only'}
{attribute 'strict'}
TYPE ePowerstate :
(
	Charging := -1,
	None := 0,
	Discharging := 1		
)INT;
END_TYPE

// ---- POUs/Objects/PowerStack/_Enums/eStatusPowerModule.TcDUT
{attribute 'qualified_only'}
{attribute 'strict'}
{attribute 'to_string'}
TYPE eStatusPowerModule :
(
	Init					:= 0,	// Not ready to do anything yet
	off						:= 1, 	// OFF MCCBs OPEN,
	DcOK					:= 2, 	// Dc voltage above 80%
	idle					:= 3, 	// MCCB CLOSED, No modulation
	running					:= 4,	// MCCB CLOSED + Modulation	
	fault					:= 10,
	EMStop					:= 11
);
END_TYPE

// ---- POUs/Objects/PowerStack/_Enums/eStatusPowerStack.TcDUT
{attribute 'qualified_only'}
{attribute 'strict'}
{attribute 'to_string'}
TYPE eStatusPowerStack :
(
	Init					:= 0,	// Not ready to do anything yet
	off						:= 1, 	// OFF MCCBs OPEN,
	idle					:= 2, 	// MCCB CLOSED, No modulation, Netcontactor CLOSED with grid OR Netcontactor OPEN + modulation with no grid
	running					:= 3,	// MCCB CLOSED + Modulation, Netcontactor CLOSED
	ecorunning				:= 4,	// MCCB CLOSED + Modulation with only one out of two inverters, Netcontactor CLOSED
	Wait_CoolingMode1		:= 20,
	Wait_HVDC				:= 21,
	Start_Master			:= 22, 	// Starting master
	Start_Slave				:= 23,	// Starting slave
	Synchronization			:= 24,
	Wait_CoolingMode2		:= 25,
	Standby					:= 9,
	Standby_GridSupply		:= 10, 	// POWERMODULE 1 + 2 off, Netcontactor Closed
	Standby_InternalSupply	:= 11,	// PowerModule 1 ON, powermodule 2 Off, Netcontactor OPEN
	shutdown				:= 12,
	fault					:= 13,
	GridCodeStop			:= 14,
	Cooling_Shutdown		:= 15  // 	
);		
END_TYPE

// ---- POUs/Objects/PowerStack/_Structs/NestedStructs/ST_InverterControlWord.TcDUT
TYPE ST_InverterControlWord :
STRUCT
	b_ChargeDC				: BOOL;
	b_run					: BOOL;
	b_Reset					: BOOL;
	b_FieldbusControlEnable	: BOOL;
	b_WatchdogPulse			: BOOL;
	b_ParallelAFE			: BOOL;
	b_PIDenable				: BOOL;
	b_GridCodeEnable		: BOOL;
	b_ExtGridcodeTrip		: BOOL;
END_STRUCT
END_TYPE

// ---- POUs/Objects/PowerStack/_Structs/NestedStructs/ST_Inverter_additionalTemperatures.TcDUT
TYPE ST_Inverter_additionalTemperatures :
STRUCT
	r_ambient					: REAL;
	r_CMchokeOuter				: ARRAY[1..4] OF REAL;
	r_CMchokeInner				: ARRAY[1..4] OF REAL;
	r_GrChokeOuter				: ARRAY[1..3] OF REAL;
	r_GrChokeInner				: ARRAY[1..3] OF REAL;
	r_ACCapsTop					: REAL;
	r_ACCapsBottom				: REAL;
	r_DCCaps					: REAL;
	r_ACbusbarOutput			: REAL;
	r_ACbusbarCMchoke			: REAL;
	r_DCbusbarCMChoke			: REAL;
	r_AirInletModule			: REAL;
	r_AirOutletFancoil			: REAL;
	r_WaterInletFancoil			: REAL;
	r_WaterOutletFancoil		: REAL;
	r_FancoilCompartement		: REAL;
END_STRUCT
END_TYPE

// ---- POUs/Objects/PowerStack/_Structs/NestedStructs/ST_Inverter_LineState.TcDUT
TYPE ST_Inverter_LineState :
STRUCT
	b_LineVoltTripLimHigh		: BOOL;
	b_LineVoltTripLimlow		: BOOL;
	b_LineFreqTripLimHigh		: BOOL;
	b_LineFreqTripLimLow		: BOOL;
	b_LineFreqOK				: BOOL;
	b_LineVoltOK				: BOOL;
	b_FRTActive					: BOOL;
	b_GridCodeTripActive		: BOOL;
END_STRUCT
END_TYPE

// ---- POUs/Objects/PowerStack/_Structs/NestedStructs/ST_Inverter_StatusWord.TcDUT
TYPE ST_Inverter_StatusWord :
STRUCT
	//General Status Word Variables
		b_ReadyToDCCharge				: BOOL;
		b_ReadyToOperate				: BOOL;
		b_Running						: BOOL;
		b_Fault							: BOOL;
		b_RunEnabled					: BOOL;
		b_QuickstopNotActive			: BOOL;
		b_MCCBControlNotOK				: BOOL;
		b_Warning						: BOOL;
		b_DCAtReference					: BOOL;
		b_DCAboveLimit					: BOOL;
		b_WatchdogFeedback				: BOOL;
END_STRUCT
END_TYPE

// ---- POUs/Objects/PowerStack/_Structs/NestedStructs/ST_Inverter_UgridStatusWord.TcDUT
TYPE ST_Inverter_UgridStatusWord :
STRUCT
	//Ugrid Status Word
		b_ChargeControlActive			: BOOL;
		b_InternalChargingSwitchStatus	: BOOL;
		b_MCBcontrol					: BOOL;
		b_MCBStatus						: BOOL;
		b_RunEnabled					: BOOL;
		b_DriveReady					: BOOL;
		b_AFEmodeActive					: BOOL;
		b_IslandModeActive				: BOOL;
		b_MicrogridModeActive			: BOOL;
		b_RunRequestActive				: BOOL;
		b_DriveInRunState				: BOOL;
		b_FaultActive					: BOOL;
		b_SynchronizedToD7				: BOOL;
		b_D7MeasurementsOK				: BOOL;	
END_STRUCT
END_TYPE

// ---- POUs/Objects/PowerStack/_Structs/NestedStructs/ST_Inverter_Write.TcDUT
TYPE ST_Inverter_Write :
STRUCT
	Controlword				: ST_InverterControlWord;
	ui_ControlwordValue		: UINT;
	i_invertermode 			: INT;
	i_BaseCurrentRef 		: INT;
	i_ReactiveCurrentRef	: INT;
	i_FrequencyDroop		: INT;
	i_VoltageDroop			: INT;
	i_FrequencyDroopOffset	: INT;
	i_VoltageCorrection		: INT;
	i_BaseRefRampRate		: INT;
	i_StartPowerMode		: INT;
	i_StartVoltageMode		: INT;
	i_OutActCurrentLimit	: INT;
	i_InActCurrentLimit		: INT;
	i_DCVramprate			: INT;
END_STRUCT
END_TYPE

// ---- POUs/Objects/PowerStack/_Structs/NestedStructs/ST_Powermodule_CalibData.TcDUT
TYPE ST_Powermodule_CalibData :
STRUCT
	Pset: ARRAY[0..4] OF REAL;
	Qset: ARRAY[0..4] OF REAL;
	Pmeas: ARRAY[0..4] OF ARRAY[0..4] OF REAL;
	Qmeas: ARRAY[0..4] OF ARRAY[0..4] OF REAL;
END_STRUCT
END_TYPE

// ---- POUs/Objects/PowerStack/_Structs/NestedStructs/ST_Powermodule_Events.TcDUT
TYPE ST_Powermodule_Events :
STRUCT
		b_GeneralFaultFlag				: BOOL;
		b_GeneralWarningFlag			: BOOL;

		//Powermodule Warnings
		b_CMSTemperatureRangeWarning	: BOOL;
		b_FanStateUnknownWarning		: BOOL;
		b_TempThrottlingActive			: BOOL;
		b_CurrThrottlingActive			: BOOL;
		
		//INVERTER Fault Status Word 
		b_F1OverCurrent					: BOOL;
		b_F2OverVoltage					: BOOL;
		b_F9UnderVoltage				: BOOL;
		b_F91ShortCircuit				: BOOL;
		b_F3EarthFault					: BOOL;
		b_Spare							: BOOL;
		b_F14UnitOverTemperature		: BOOL;
		b_F56TemperatureFault			: BOOL;
		b_F10LineSynchFault				: BOOL;
		b_F52KeypadOCCommFault			: BOOL;
		b_F53FieldbusFault				: BOOL;
		b_F59SystembusFault				: BOOL;
		b_F54SlotCommunicationFault		: BOOL;
		b_F50Meas4mAFault				: BOOL;
		b_F11OutputPhaseFault 			: BOOL;
		b_F80ChargeFault				: BOOL;
		b_F51ExternalFault				: BOOL;
		b_F31IGBTFault					: BOOL;
		b_F64MCBstateFault				: BOOL;
		b_WatchdogError					: BOOL;
		b_24VdcUVRFault					: BOOL;
		
		//Buscoupler connected faults
		b_MCCBtrip						: BOOL;	
		b_ShutdownTimeOut				: BOOL;
		b_StartUpTimeOut				: BOOL;
	
		//Temperature faults and warnings 
		b_CMChokeTemperatureHigh		: ARRAY [1..4] OF BOOL;
		b_CMChokeTemperatureTooHigh		: ARRAY [1..4] OF BOOL;
		b_GridChokeTemperatureHigh		: ARRAY [1..3] OF BOOL;
		b_GridChokeTemperatureTooHigh	: ARRAY [1..3] OF BOOL;
		b_inverterTemperatureHigh		: BOOL;
		b_PT100Overrange				: BOOL;
		b_PT100Underrange				: BOOL;
		by_PT100ErrorCount				: BYTE;
		

		
END_STRUCT
END_TYPE

// ---- POUs/Objects/PowerStack/_Structs/NestedStructs/ST_Powermodule_PowerCurveCoefficients.TcDUT
TYPE ST_Powermodule_PowerCurveCoefficients :
STRUCT
	enable: BOOL;
	a : REAL;
	b : REAL;
	c : REAL;
	d : REAL; 
	e : REAL;
	f : REAL;
END_STRUCT
END_TYPE

// ---- POUs/Objects/PowerStack/_Structs/NestedStructs/ST_PowerStack_Events.TcDUT
TYPE ST_PowerStack_Events :
STRUCT
	//INFO
	b_CoolingDerating				: BOOL;
	b_PlimitShiftingActive			: BOOL;
	
	//Warnings
	b_DCdeviationHigh				: BOOL;
	b_TemperatureWarning			: BOOL;
	b_OvercurrentWarning			: BOOL;
	b_UndervoltageWarning			: BOOL;
	b_OvervoltageWarning			: BOOL;
	b_TemperatureDeviationHigh		: BOOL;
	b_PlimitShutdownWarning			: BOOL;
	
	b_MasterWarning					: BOOL;
	b_SlaveWarning					: BOOL;
	b_GridCodeWarning				: BOOL;
	
	//faults
	b_UnderFreqFault				: BOOL;
	b_OverFreqFault					: BOOL;
	b_UnderVoltageFault				: BOOL;
	b_OverVoltageFault				: BOOL;
	b_OvercurrentFault				: BOOL;
	b_PlimitShutdown				: BOOL;
	b_TemperatureFault				: BOOL;
	b_MasterFault					: BOOL;
	b_SlaveFault					: BOOL;
	b_NetcontactorFault				: BOOL;
	
	
	b_startupTimeOut				: BOOL;
	b_ShutdownTimeOut				: BOOL;
	
	ui_shutdownRemainingTime		: UINT;
END_STRUCT
END_TYPE

// ---- POUs/Objects/PowerStack/_Structs/NestedStructs/ST_Powerstack_ShiftingParams.TcDUT
TYPE ST_Powerstack_ShiftingParams :
STRUCT
	InitialOverloadDelay		: TIME := T#1S; // ignore initial power surge
	ShutdownDelay				: TIME := T#1M; // shutdown delay when limit is exceeded.
	ShiftingHoldTime			: TIME := T#20M; // when shifting is applied, this time must pass before returning back.
	ShiftingRate				: TIME := T#100MS; // time per step. Number of steps is + and - 1000. The stepsize is 1/2000 of the set min / max range.
	FreqMaxPu					: REAL := 1.03; //per unit
	FreqMinPu					: REAL := 0.97;
	VoltMaxPu					: REAL := 1.1;
	VoltMinPu					: REAL := 0.9;
END_STRUCT
END_TYPE

// ---- POUs/Objects/PowerStack/_Structs/ST_PowerModule_calibration.TcDUT
TYPE ST_PowerModule_calibration :
STRUCT
	b_StartCalibration			: BOOL;
	r_Pset						: REAL;
	r_Qset						: REAL;
	PCoefficients				: ST_Powermodule_PowerCurveCoefficients;
	QCoefficients				: ST_Powermodule_PowerCurveCoefficients;
	CalibrationData				: ST_Powermodule_calibData;
END_STRUCT
END_TYPE

// ---- POUs/Objects/PowerStack/_Structs/ST_PowerModule_get.TcDUT
TYPE ST_PowerModule_get :
STRUCT
	b_online						: BOOL;

	r_ApparentPower					: REAL;
	r_ActivePower					: REAL;
	r_ReactivePower					: REAL;
	r_ACVoltageD7					: REAL;
	r_VoltageDroop					: REAL;
	r_ACVoltageSupply				: REAL;
	r_FrequencyD7					: REAL;
	r_FrequencyDroop				: REAL;
	r_FrequencySupply				: REAL;
	r_CurrentUnbalance				: REAL;
	r_DCPower						: REAL;
	r_DCVoltage						: REAL;
	r_DCCurrent						: REAL;
	r_ACCurrent						: REAL;
	r_ActiveCurrent					: REAL;
	r_ReactiveCurrent				: REAL;
	r_LoadPercent					: REAL; //%
	r_D7SyncError					: REAL;
	r_Pmin							: REAL;
	r_Pmax							: REAL;
	r_QMax							: REAL;
	r_Qmin							: REAL;
	r_Pset							: REAL;
	r_Qset							: REAL;
	r_ACcurrentLimit				: REAL; 
	r_OverCurrentValue				: REAL; // overcurrent ratio 0 .. 1.25 x rated current
	r_ModulationIndex				: REAL;
	
	r_TemperatureInverter			: REAL;
	r_TemperatureGridChoke			: ARRAY [1..3] OF REAL;
	r_TemperatureCMChoke			: ARRAY [1..4] OF REAL;
	r_TemperatureMax				: REAL;
	AddTemperatures					: ST_Inverter_additionalTemperatures;
	w_TemperatureFaultWord			: WORD;
	w_OperationHours				: WORD;
	
	e_PowerMode						: ePowerModes;
	e_InverterMode					: eInverterModes;
	e_Status						: eStatusPowermodule;
	e_ThrottlingStatus					: ePowerModuleThrottlingState;		
	ui_InverterCommStatus			: UINT;
	ui_BuscouplerCommStatus			: UINT;
	
	b_MccbTripOK					: BOOL;
	b_MccbUvr24VdcOK				: BOOL;
	b_MccbFb						: BOOL;
	b_FanFb							: BOOL;
	b_DCcontactorFb					: BOOL;
	b_PrechargeContactor			: BOOL;
	b_LimiterActive					: BOOL;
	eConditioningRequirement		: eConditioningRequirement;
	b_FlowSwitchOK					: Bool;
	
	StatusWord						: ST_Inverter_StatusWord;
	UgridStatusWord					: ST_Inverter_UgridStatusWord;
	GridcodeStatusWord				: ST_Inverter_LineState;
	Events							: ST_Powermodule_Events;
	controldata						: ST_Inverter_write;
	
END_STRUCT
END_TYPE

// ---- POUs/Objects/PowerStack/_Structs/ST_PowerModule_params.TcDUT
TYPE ST_PowerModule_params :
STRUCT
	//Rated settings
	r_InverterRatedCurrent			: REAL := 460; //Ampere // according danfoss grid current rating
	r_InverterRatedPower			: REAL := 360; //kva // according rated max current
	i_VoltageOffset					: INT := 4; //correction factor voltage control.
	i_DCVramprate					: INT := -1; //-1 = disabled
	
	//Limits
	r_ACCurrentLimitMax				: REAL := 650;
	r_ACcurrentLimitMin				: REAL := 100;
	r_ModulationIndexLimit			: REAL := 98; //indicator for AC voltage limitation of the drive. Controls AC limit PID.
	r_ModulationIndexLimitHyst		: REAL := 0.5; 
	
	//Temperatures and conditioning
	r_powerLoadFanOn				: REAL := 30;	
	r_FilterTempFanOn				: REAL := 50;
	r_FilterTempWarning				: REAL := 80; //also used for throttling start
	r_FilterTempAlarm				: REAL := 90; //also used for for throttling end 
	r_InverterTempWarning			: REAL := 55; //also used for throttling start
	r_InverterTempAlarm				: REAL := 60; //also used for for throttling end 
	r_ThrottlingMinimum				: REAL := 0.3; //% of rated power.
	
	//Releases
	ui_DCVoltageDeltaPrechargeOK	: UINT := 20; // VDC
	ui_DCvoltageMinPrechargeOK		: UINT := 590; //VDC
	
END_STRUCT
END_TYPE

// ---- POUs/Objects/PowerStack/_Structs/ST_PowerModule_set.TcDUT
TYPE ST_PowerModule_set :
STRUCT
	//commands
	b_RunEnable						: BOOL;
	r_ActivePower					: REAL;
	r_ReactivePower					: REAL;
	r_NomFrequency					: REAL;
	r_NomVoltage					: REAL;
	r_FrequencyDroop				: REAL;
	r_VoltageDroop					: REAL;
	r_Pmax							: REAL;
	r_Pmin							: REAL;
	r_ACcurrentLimit				: REAL;
	i_PowerChangeRate				: INT; // % nominal power / s
	r_overcurrentFactor				: REAL;
	r_DroopMinimum					: REAL := 0.1;
	r_DroopIslandMode				: REAL := 0.1;
	r_DroopMaximum					: REAL := 10; //%
	
	//WRITE DATA Buscoupler
	b_FanContactor					: BOOL;
	b_D7SyncRequest					: BOOL;
	b_QuickstopInactive				: BOOL;
	b_gridcodeEnable				: BOOL;
	b_ExtgridCodeTrip				: BOOL;
END_STRUCT
END_TYPE

// ---- POUs/Objects/PowerStack/_Structs/ST_Powerstack_Calibration.TcDUT
TYPE ST_Powerstack_Calibration:
STRUCT
	Master				: ST_PowerModule_calibration;
	Slave				: ST_PowerModule_calibration;
END_STRUCT
END_TYPE

// ---- POUs/Objects/PowerStack/_Structs/ST_PowerStack_get.TcDUT
TYPE ST_PowerStack_get :
STRUCT
	// ENUMS
	e_State							: eStatusPowerStack;
	e_PowerState					: ePowerstate;
	e_InverterMode					: eInverterModes;			//0=AFE, Micro, Island, transition
	e_PowerMode						: ePowerModes;				//0=IsoChronous, 1= Droop
	e_ThrottlingStatus				: ePowerModuleThrottlingState;
	
	//POWER DATA (REALS)
	r_VoltageDroop					: REAL;				
	r_FrequencyDroop				: REAL;
	r_ACVoltageD7					: REAL; 
	r_FrequencyD7					: REAL; 
	r_ActivePower					: REAL;
	r_ReactivePower					: REAL;
	r_Pmin							: REAL;
	r_Pmax							: REAL; 
	r_QMax							: REAL;
	r_QMin							: REAL;	
	r_Smax							: REAL;
	r_ACcurrentLimit				: REAL;
	r_ACcurrentLimitMax				: REAL;
	r_PowerChangeRate				: REAL;
	r_ApparentPower					: REAL;
	r_CosPhi						: REAL;
	r_AcCurrent						: REAL;
	r_DCPower						: REAL;
	r_DCVoltage						: REAL;
	r_DCcurrent						: REAL;
	r_ACVoltageSupply				: REAL;
	r_FrequencySupply				: REAL;
	r_LoadPercent					: REAL; //%
	r_RatedCurrent					: REAL;
	r_RatedPower					: REAL;
	r_OvercurrentValueAct			: REAL; //actual overcurrent value
	r_OvercurrentValueMax			: REAL; //max overcurrent value
	r_ThrottlingValueAct			: REAL; // %percentage , inverse of overcurrent with 100%
	
	//Booleans
	b_GridTied						: BOOL;
	b_GridCodeCheckActive			: BOOL;
	b_GridCodeOK					: BOOL := TRUE;
	b_GridACdetected				: BOOL;
	b_InverterGridFormingMode		: BOOL;
	b_ACDetected					: BOOL;
	b_DCDetected					: BOOL;
	b_InverterRunning				: BOOL;
	b_StartedState					: BOOL;
	b_ControlEnabled				: BOOL;
	b_EcomodeAvailable				: BOOL;
	b_StartEnabled					: BOOL;				

	//Temperatures
	r_MaxTemperature				: REAL;
	
	//timers
	t_ShiftHoldTimeRemaining		: TIME;
	t_GridCodeReconnectTime			: TIME;
	//structs
	Events							: ST_PowerStack_Events;
	
	//Sublevel data
	PowermoduleMaster				: REFERENCE TO ST_PowerModule_get();
	PowermoduleSlave				: REFERENCE TO ST_PowerModule_get();
	Netcontactor					: REFERENCE TO ST_Netcontactor_get();
	
END_STRUCT
END_TYPE

// ---- POUs/Objects/PowerStack/_Structs/ST_Powerstack_LOMParams.TcDUT
TYPE ST_Powerstack_LOMParams :
STRUCT
	ForceSlowDetection	: BOOL := FALSE;
	FreqFilterLength	: UINT := 5; // samples 
	DetectionTimeFast_ms: UINT := 50; // milliseconds
	DetectionTimeSlow_ms: UINT := 1000; // milliseconds
	RoCofLimit			: REAL := 0.5; // Hz/s
	PowerPulseSize		: REAL := 0.5; // %, of rated power during ugrid to enable LOM detection.
	EnablePowerPulse	: BOOL := TRUE;
END_STRUCT
END_TYPE

// ---- POUs/Objects/PowerStack/_Structs/ST_PowerStack_params.TcDUT
TYPE ST_PowerStack_params :
STRUCT
	b_RunEnable				: BOOL := TRUE; //enable inverter run 
	b_StandbyEnable			: BOOL := TRUE;
	b_GridcodesEnabled		: BOOL := TRUE;
	r_DroopMinimum			: REAL := 0.0;
	r_DroopIslandMode		: REAL := 0.1;
	r_DroopMaximum			: REAL := 10; //%
	r_ReactiveOffset		: REAL := 0;
	ui_DeratingStack		: UINT := 5; // %
	ui_DeratingLimCooling	: UINT := 80; // %
	i_MaxPowerChangeRate	: INT := 500; // %/s
	ui_OvercurrentRating	: UINT := 150; // %
	i_ChargeOnlyIdlePower	: INT := -3;
	r_ActiveSetpointGain	: REAL := 1; 
	r_ReactiveSetpointGain  : REAL := 1;
	
	//AC drive limits
	r_FreqLowLimit			: REAL := 48;
	r_FreqHighLimit			: REAL := 52; 
	ui_FreqLimitTripDelay	: UINT := 2000; // milliseconds
	FreqVoltageShift		: st_powerstack_ShiftingParams;
	
	PowermoduleMaster		: ST_PowerModule_params;
	PowermoduleSlave		: ST_PowerModule_params;
	LOM						: ST_Powerstack_LOMParams;
END_STRUCT
END_TYPE

// ---- POUs/Objects/PowerStack/_Structs/ST_PowerStack_Set.TcDUT
TYPE ST_PowerStack_Set :
STRUCT
	//WRITE
	b_NetcontactorHoldClose			: BOOL; // used when input breaker or external PSB breaker must be controlled instead of netcontactor.
	b_ExtGridConnected				: BOOL;
	b_DisableShifting				: BOOL;
	b_slowLom						: BOOL;
	b_automaticswitching			: BOOL;
	b_GridCodeEnable				: BOOL := TRUE;
	e_InverterMode					: eInverterModes;			//0=AFE, 1= ugrid, 2, island
	e_PowerMode						: ePowerModes;				//
	e_NetconClosingRequest			: eNetcontMode;
	e_PowerLimitingMode				: ePLM;
	r_VoltageDroop					: REAL;				
	r_FrequencyDroop				: REAL;
	r_NominalOutputVoltage			: REAL := 400; //R/W
	r_NominalOutputFrequency		: REAL := 50; //R/W
	r_ActivePower					: REAL; //R/W
	r_ReactivePower					: REAL; //R/W
	
	//limits
	r_Pmax							: REAL;
	r_Pmin							: REAL;
	r_ACcurrentLimit				: REAL;
	
END_STRUCT
END_TYPE

// ---- POUs/Objects/ProtectionSystems/FireDetection/_Enums/eCOAlarmStatus.TcDUT
{attribute 'qualified_only'}
{attribute 'strict'}
{attribute 'tostring'}
TYPE eCOAlarmStatus :
(
	Error			:= 0,
	Normal 			:= 1,
	WarningLevel1 	:= 2,
	WarningLevel2 	:= 3,
	Alarm 			:= 4
);
END_TYPE

// ---- POUs/Objects/ProtectionSystems/FireDetection/_Enums/eSmokeDetectAlarmStatus.TcDUT
{attribute 'qualified_only'}
{attribute 'strict'}
{attribute 'tostring'}
TYPE eSmokeDetectAlarmStatus :
(
	Error := 0,
	Normal := 1,
	Alarm := 2
);
END_TYPE

// ---- POUs/Objects/ProtectionSystems/FireDetection/_Structs/ST_CODetectors.TcDUT
TYPE ST_CODetectors :
STRUCT
	State 			: 	eCOAlarmStatus;
	b_CoValuesOK	: 	BOOL;
	Value 			:  	ARRAY[0..3] OF REAL;	//-1 if inoperative. [0]=mean [1]=CO1 [2]=CO2 [3]=max
END_STRUCT
END_TYPE

// ---- POUs/Objects/ProtectionSystems/FireDetection/_Structs/ST_FireDetection_get.TcDUT
TYPE ST_FireDetection_get :
STRUCT
	b_FireAlarm		: 	BOOL;
	SmokeDetectors 	:	ST_SmokeDetectors;
	CODetectors		:	ST_CODetectors;
	Events			:	ST_FireSystem_Events;
END_STRUCT
END_TYPE

// ---- POUs/Objects/ProtectionSystems/FireDetection/_Structs/st_Firedetection_params.TcDUT
TYPE st_Firedetection_params :
STRUCT
	r_COwarningLevel_1				: REAL := 10;
	r_COwarningLevel_2				: REAL := 20;
	r_COalarmLevel					: REAL := 120;
	r_COrange						: REAL := 500;
END_STRUCT
END_TYPE

// ---- POUs/Objects/ProtectionSystems/FireDetection/_Structs/ST_FireDetection_set.TcDUT
TYPE ST_FireDetection_set :
STRUCT
	SilenceSounder	:	BOOL; //only disables currently activated alarm.
	TestSounder		:	BOOL;
END_STRUCT
END_TYPE

// ---- POUs/Objects/ProtectionSystems/FireDetection/_Structs/ST_FireSystem_Events.TcDUT
TYPE ST_FireSystem_Events :
STRUCT
	CODetFault		:	BOOL;
	CODetWarning1	:	BOOL;
	CODetWarning2	: 	BOOL;
	CODetAlarm		:	BOOL;
	SmokeDetFault	:	BOOL;
	SmokeDetAlarm	:	BOOL;
	AlarmMuted		:	BOOL;
END_STRUCT
END_TYPE

// ---- POUs/Objects/ProtectionSystems/FireDetection/_Structs/ST_SmokeDetectors.TcDUT
TYPE ST_SmokeDetectors :
STRUCT
	State : eSmokeDetectAlarmStatus;
END_STRUCT
END_TYPE

// ---- POUs/Objects/ProtectionSystems/FireDetection/_Structs/ST_SmokeDetIO.TcDUT
TYPE ST_SmokeDetIO :
STRUCT
	Signal_OK 	: BOOL;
	Power_OK 	: BOOL;
END_STRUCT
END_TYPE

// ---- POUs/Objects/ProtectionSystems/InsulationMonitoring/_Structs/ST_InsulationMonitor_get.TcDUT
TYPE ST_InsulationMonitor_get :
STRUCT
	b_Enabled							: BOOL;	
	b_PENlinkDetected					: BOOL;
	b_Warning							: BOOL;
	e_EarthingSystemDetected			: eEarthingSystems;
	b_PENlinkOperatedFault				: BOOL;
	b_EarthingSystemMismatch			: BOOL;
	b_NoEarthingSystemSet				: BOOL;
END_STRUCT
END_TYPE

// ---- POUs/Objects/ProtectionSystems/InsulationMonitoring/_Structs/ST_InsulationMonitor_params.TcDUT
TYPE ST_InsulationMonitor_params :
STRUCT
	i_EarthSystemDetectionDelay		:INT := 60; // Seconds
END_STRUCT
END_TYPE

// ---- POUs/Objects/ProtectionSystems/InsulationMonitoring/_Structs/St_InsulationMonitor_PassThrough.TcDUT
TYPE St_InsulationMonitor_PassThrough :
STRUCT
	b_NetContFB				: BOOL;
	b_MccbfbMaster			: BOOL;
	b_MccbfbSlave			: BOOL;
	b_ACdetected			: BOOL;
	b_PENlinkFB				: BOOL;	
END_STRUCT
END_TYPE

// ---- POUs/Objects/ProtectionSystems/InsulationMonitoring/_Structs/ST_InsulationMonitor_set.TcDUT
TYPE ST_InsulationMonitor_set :
STRUCT
	b_enable			: BOOL;
 	e_EarthingSystem	: eEarthingSystems := eEarthingSystems.TN;
END_STRUCT
END_TYPE

// ---- POUs/Objects/ProtectionSystems/OvercurrentProtection/_Structs/ST_OvercurrentProtection_Events.TcDUT
TYPE ST_OvercurrentProtection_Events :
STRUCT
	Input	:ARRAY [1..2] OF ARRAY [1..4] OF FB_Overcurrentdetect(); //FB_UpperLimitAndTimeExceeded();
	Output	:ARRAY [1..3] OF ARRAY [1..4] OF FB_Overcurrentdetect();
END_STRUCT
END_TYPE

// ---- POUs/Objects/ProtectionSystems/OvercurrentProtection/_Structs/ST_OvercurrentProtection_get.TcDUT
TYPE ST_OvercurrentProtection_get :
STRUCT
	//Overcurrent Powerlocks
	r_TotalOutputCurrentLimit			: REAL := 0;
	r_TotalInputCurrentLimit			: REAL := 0;
	b_OutputWarning						: BOOL;
	b_InputWarning						: BOOL;
	b_OutputAlarm						: BOOL;
	b_InputAlarm						: BOOL;
	r_PeakCurrent						: REAL;
	t_PeakCurrentDuration				: TIME;
	s_locationPeak						: STRING;
	
	Events								: ST_OvercurrentProtection_events;
END_STRUCT
END_TYPE

// ---- POUs/Objects/ProtectionSystems/OvercurrentProtection/_Structs/ST_OvercurrentProtection_InternalLinking.TcDUT
TYPE ST_OvercurrentProtection_InternalLinking :
STRUCT
	a_r_CurrentInput			: ARRAY [1..2] OF ARRAY[1..4] OF REAL; //first array of powerlockset, second of powerlock
	a_r_CurrentOutput			: ARRAY [1..3] OF ARRAY[1..4] OF REAL;
	b_InputSectionAvailable 	: BOOL;
	b_thirdOutputAvailable 		: BOOL;
END_STRUCT
END_TYPE

// ---- POUs/Objects/ProtectionSystems/OvercurrentProtection/_Structs/ST_OvercurrentProtection_Params.TcDUT
TYPE ST_OvercurrentProtection_Params :
STRUCT
	ui_OCPtripTime		: UINT := 900; //Seconds
	ui_Ik				: UINT := 16; // Short circuit capacity of component to be protected [Ik/s]
	ui_Irated			: UINT := 400; // rated current 
	ui_gain				: UINT := 10; //gain for tuning calculated remaining time during overcurrent.
	OutputNormalShutdownDelay : TIME := T#5S;
END_STRUCT
END_TYPE

// ---- POUs/Objects/ProtectionSystems/OvercurrentProtection/_Structs/ST_OvercurrentProtection_set.TcDUT
TYPE ST_OvercurrentProtection_set :
STRUCT
	ui_PowerlockInputCurrentLimit			: ARRAY [1..2] OF UINT := [400,400];
	ui_PowerlockOutputCurrentLimit			: ARRAY [1..3] OF UINT := [400,400,400];
END_STRUCT
END_TYPE

// ---- POUs/Objects/ProtectionSystems/ResidualCurrentMonitoring/_Structs/ST_ResidualCurrentMonitor_get.TcDUT
TYPE ST_ResidualCurrentMonitor_get :
STRUCT
	b_prewarning			: BOOL;
END_STRUCT
END_TYPE

// ---- POUs/Objects/ProtectionSystems/SurgeProtection/_Structs/ST_Surgeprotection_get.TcDUT
TYPE ST_Surgeprotection_get :
STRUCT
	b_Type12_OK				: BOOL;
	b_Type3_OK				: BOOL;			
END_STRUCT
END_TYPE

// ---- POUs/Objects/ProtectionSystems/_Struct/ST_ProtectionSystems_get.TcDUT
TYPE ST_ProtectionSystems_get :
STRUCT
	//Fire Detection System
	FireDetection						: ST_Firedetection_get;
	
	//InsulationMonitor
	Insulation							: ST_InsulationMonitor_get;
	
	//MRCDB
	MRCDB								: ST_ResidualCurrentMonitor_get;
	
	//Surge protection
	Surge								: ST_SurgeProtection_get;
	
	//Overcurrent protection
	OvercurrentProtection				: ST_OverCurrentProtection_Get;
	
END_STRUCT
END_TYPE

// ---- POUs/Objects/ProtectionSystems/_Struct/ST_ProtectionSystems_Params.TcDUT
TYPE ST_ProtectionSystems_Params :
STRUCT
	InsulationMonitor				: ST_InsulationMonitor_params;
	firedetection					: ST_Firedetection_params;
	OCP								: ST_Overcurrentprotection_params;
END_STRUCT
END_TYPE

